C05419=1052.295,341.626,-112.495,173.245,38.864,157.407
C05420=1052.302,341.873,-112.531,173.249,38.868,157.408
C05421=1052.309,342.120,-112.568,173.254,38.872,157.409
C05422=1052.316,342.368,-112.604,173.258,38.877,157.410
C05423=1052.322,342.616,-112.640,173.262,38.881,157.411
C05424=1052.330,342.863,-112.676,173.267,38.886,157.413
C05425=1052.337,343.109,-112.713,173.271,38.890,157.414
C05426=1052.344,343.357,-112.749,173.276,38.894,157.415
C05427=1052.351,343.604,-112.786,173.280,38.899,157.416
C05428=1052.358,343.851,-112.822,173.284,38.904,157.417
C05429=1052.365,344.098,-112.858,173.289,38.908,157.418
C05430=1052.372,344.346,-112.894,173.293,38.913,157.419
C05431=1052.379,344.593,-112.931,173.298,38.917,157.421
C05432=1052.386,344.841,-112.968,173.302,38.921,157.422
C05433=1052.393,345.088,-113.004,173.306,38.926,157.423
C05434=1052.400,345.335,-113.041,173.312,38.931,157.424
C05435=1052.407,345.582,-113.078,173.316,38.935,157.425
C05436=1052.414,345.829,-113.114,173.321,38.939,157.426
C05437=1052.421,346.077,-113.151,173.325,38.944,157.428
C05438=1052.429,346.355,-113.192,173.330,38.949,157.429
C05439=1052.437,346.633,-113.233,173.335,38.954,157.430
C05440=1052.444,346.912,-113.275,173.340,38.959,157.432
C05441=1052.454,347.190,-113.316,173.346,38.964,157.433
C05442=1052.460,347.437,-113.353,173.350,38.969,157.434
C05443=1052.467,347.685,-113.390,173.355,38.973,157.435
C05444=1052.474,347.932,-113.427,173.359,38.978,157.437
C05445=1052.481,348.179,-113.463,173.364,38.982,157.438
C05446=1052.489,348.426,-113.501,173.368,38.987,157.439
C05447=1052.495,348.674,-113.537,173.373,38.992,157.440
C05448=1052.503,348.920,-113.574,173.377,38.996,157.441
C05449=1052.510,349.168,-113.611,173.382,39.001,157.443
C05450=1052.517,349.415,-113.648,173.386,39.005,157.444
C05451=1052.524,349.663,-113.685,173.391,39.010,157.445
C05452=1052.532,349.910,-113.722,173.396,39.015,157.446
C05453=1052.539,350.156,-113.759,173.401,39.019,157.447
C05454=1052.545,350.404,-113.796,173.405,39.024,157.449
C05455=1052.553,350.651,-113.834,173.410,39.028,157.450
C05456=1052.561,350.898,-113.870,173.414,39.033,157.451
C05457=1052.568,351.145,-113.907,173.419,39.038,157.452
C05458=1052.574,351.392,-113.944,173.423,39.043,157.453
C05459=1052.582,351.639,-113.982,173.429,39.047,157.455
C05460=1052.589,351.886,-114.019,173.433,39.052,157.456
C05461=1052.596,352.134,-114.056,173.438,39.057,157.457
C05462=1052.603,352.381,-114.094,173.443,39.062,157.458
C05463=1052.610,352.628,-114.131,173.447,39.066,157.460
C05464=1052.617,352.875,-114.168,173.452,39.071,157.461
C05465=1052.624,353.122,-114.206,173.456,39.076,157.462
C05466=1052.631,353.369,-114.244,173.462,39.081,157.463
C05467=1052.639,353.616,-114.281,173.466,39.086,157.465
C05468=1052.646,353.863,-114.319,173.471,39.090,157.466
C05469=1052.653,354.110,-114.356,173.476,39.095,157.467
C05470=1052.660,354.357,-114.394,173.480,39.100,157.468
C05471=1052.668,354.605,-114.431,173.485,39.105,157.470
C05472=1052.675,354.852,-114.469,173.490,39.109,157.471
C05473=1052.682,355.099,-114.506,173.495,39.114,157.472
C05474=1052.689,355.346,-114.544,173.500,39.119,157.474
C05475=1052.697,355.593,-114.581,173.504,39.124,157.475
C05476=1052.703,355.840,-114.618,173.509,39.129,157.476
C05477=1052.711,356.087,-114.656,173.515,39.134,157.477
C05478=1052.719,356.334,-114.695,173.519,39.139,157.479
C05479=1052.726,356.581,-114.732,173.524,39.144,157.480
C05480=1052.733,356.828,-114.770,173.529,39.148,157.481
C05481=1052.740,357.075,-114.807,173.534,39.153,157.483
C05482=1052.748,357.322,-114.845,173.539,39.158,157.484
C05483=1052.755,357.569,-114.883,173.544,39.163,157.485
C05484=1052.762,357.816,-114.920,173.548,39.168,157.486
C05485=1052.769,358.063,-114.959,173.553,39.173,157.488
C05486=1052.776,358.310,-114.997,173.559,39.178,157.489
C05487=1052.784,358.557,-115.034,173.563,39.183,157.490
C05488=1052.791,358.804,-115.073,173.568,39.188,157.492
C05489=1052.798,359.051,-115.110,173.573,39.193,157.493
C05490=1052.805,359.298,-115.149,173.579,39.198,157.494
C05491=1052.812,359.545,-115.186,173.583,39.203,157.496
C05492=1052.821,359.792,-115.225,173.588,39.208,157.497
C05493=1052.828,360.039,-115.263,173.593,39.213,157.498
C05494=1052.836,360.323,-115.307,173.599,39.219,157.500
C05495=1052.845,360.606,-115.350,173.604,39.224,157.501
C05496=1052.853,360.890,-115.394,173.611,39.230,157.503
C05497=1052.861,361.174,-115.438,173.616,39.236,157.505
C05498=1052.869,361.420,-115.477,173.621,39.241,157.506
C05499=1052.876,361.667,-115.515,173.627,39.246,157.507
C05500=1052.883,361.914,-115.553,173.631,39.251,157.509
C05501=1052.891,362.161,-115.591,173.636,39.257,157.510
C05502=1052.899,362.408,-115.630,173.642,39.262,157.511
C05503=1052.905,362.655,-115.669,173.647,39.267,157.513
C05504=1052.913,362.901,-115.707,173.651,39.272,157.514
C05505=1052.920,363.148,-115.744,173.657,39.277,157.516
C05506=1052.928,363.396,-115.784,173.662,39.282,157.517
C05507=1052.935,363.642,-115.822,173.667,39.287,157.518
C05508=1052.942,363.889,-115.861,173.673,39.293,157.520
C05509=1052.950,364.136,-115.899,173.677,39.298,157.521
C05510=1052.957,364.383,-115.938,173.682,39.303,157.523
C05511=1052.965,364.630,-115.976,173.688,39.309,157.524
C05512=1052.971,364.877,-116.015,173.693,39.314,157.525
C05513=1052.980,365.124,-116.054,173.698,39.319,157.527
C05514=1052.986,365.371,-116.093,173.704,39.324,157.528
C05515=1052.994,365.617,-116.132,173.708,39.330,157.530
C05516=1053.002,365.864,-116.171,173.713,39.335,157.531
C05517=1053.008,366.111,-116.210,173.719,39.340,157.533
C05518=1053.016,366.357,-116.248,173.724,39.346,157.534
C05519=1053.023,366.605,-116.287,173.730,39.351,157.535
C05520=1053.031,366.851,-116.326,173.735,39.356,157.537
C05521=1053.039,367.098,-116.365,173.740,39.362,157.538
C05522=1053.045,367.345,-116.404,173.746,39.367,157.540
C05523=1053.053,367.592,-116.442,173.751,39.373,157.541
C05524=1053.061,367.839,-116.482,173.755,39.378,157.543
C05525=1053.068,368.085,-116.520,173.761,39.383,157.544
C05526=1053.076,368.332,-116.560,173.766,39.389,157.546
C05527=1053.084,368.579,-116.599,173.772,39.394,157.547
C05528=1053.091,368.826,-116.638,173.777,39.399,157.549
C05529=1053.098,369.072,-116.677,173.782,39.405,157.550
C05530=1053.106,369.319,-116.716,173.788,39.410,157.551
C05531=1053.113,369.566,-116.756,173.793,39.415,157.553
C05532=1053.121,369.813,-116.795,173.799,39.421,157.555
C05533=1053.129,370.060,-116.834,173.804,39.427,157.556
C05534=1053.136,370.307,-116.873,173.810,39.432,157.557
C05535=1053.144,370.553,-116.912,173.815,39.437,157.559
C05536=1053.152,370.799,-116.952,173.821,39.443,157.561
C05537=1053.159,371.047,-116.991,173.826,39.449,157.562
C05538=1053.167,371.294,-117.030,173.831,39.454,157.563
C05539=1053.175,371.540,-117.070,173.837,39.460,157.565
C05540=1053.182,371.787,-117.109,173.842,39.465,157.567
C05541=1053.189,372.033,-117.149,173.848,39.471,157.568
C05542=1053.197,372.280,-117.189,173.853,39.477,157.570
C05543=1053.205,372.527,-117.228,173.859,39.482,157.571
C05544=1053.212,372.773,-117.267,173.864,39.488,157.573
C05545=1053.220,373.020,-117.307,173.870,39.494,157.574
C05546=1053.228,373.268,-117.347,173.875,39.500,157.576
C05547=1053.235,373.514,-117.386,173.881,39.505,157.577
C05548=1053.242,373.761,-117.426,173.886,39.511,157.579
C05549=1053.250,374.008,-117.466,173.892,39.517,157.581
C05550=1053.259,374.310,-117.515,173.899,39.524,157.582
C05551=1053.269,374.611,-117.564,173.906,39.531,157.584
C05552=1053.278,374.914,-117.613,173.913,39.538,157.586
C05553=1053.287,375.216,-117.662,173.919,39.544,157.588
C05554=1053.294,375.463,-117.702,173.925,39.550,157.590
C05555=1053.302,375.710,-117.742,173.932,39.556,157.591
C05556=1053.310,375.957,-117.781,173.937,39.562,157.593
C05557=1053.318,376.204,-117.821,173.943,39.568,157.595
C05558=1053.325,376.449,-117.862,173.948,39.574,157.596
C05559=1053.333,376.696,-117.902,173.954,39.580,157.598
C05560=1053.341,376.943,-117.941,173.960,39.586,157.599
C05561=1053.349,377.189,-117.982,173.965,39.591,157.601
C05562=1053.357,377.436,-118.021,173.972,39.597,157.603
C05563=1053.365,377.683,-118.061,173.977,39.603,157.604
C05564=1053.373,377.929,-118.102,173.983,39.609,157.606
C05565=1053.380,378.176,-118.142,173.989,39.615,157.608
C05566=1053.388,378.422,-118.182,173.994,39.621,157.609
C05567=1053.396,378.669,-118.222,174.000,39.627,157.611
C05568=1053.404,378.915,-118.263,174.006,39.633,157.613
C05569=1053.411,379.162,-118.303,174.012,39.639,157.614
C05570=1053.419,379.409,-118.344,174.018,39.645,157.616
C05571=1053.426,379.655,-118.384,174.023,39.650,157.617
C05572=1053.434,379.902,-118.424,174.030,39.656,157.619
C05573=1053.442,380.149,-118.464,174.036,39.663,157.621
C05574=1053.450,380.395,-118.505,174.041,39.668,157.622
C05575=1053.458,380.641,-118.546,174.047,39.675,157.624
C05576=1053.465,380.888,-118.587,174.054,39.681,157.626
C05577=1053.473,381.134,-118.628,174.059,39.687,157.628
C05578=1053.481,381.381,-118.667,174.065,39.693,157.629
C05579=1053.488,381.628,-118.709,174.071,39.699,157.631
C05580=1053.497,381.874,-118.749,174.078,39.706,157.633
C05581=1053.505,382.120,-118.790,174.083,39.711,157.634
C05582=1053.512,382.367,-118.831,174.089,39.718,157.636
C05583=1053.520,382.613,-118.872,174.095,39.724,157.638
C05584=1053.528,382.860,-118.913,174.101,39.731,157.640
C05585=1053.536,383.107,-118.954,174.107,39.736,157.641
C05586=1053.544,383.353,-118.995,174.113,39.743,157.643
C05587=1053.552,383.599,-119.035,174.120,39.749,157.645
C05588=1053.559,383.846,-119.077,174.125,39.755,157.647
C05589=1053.567,384.092,-119.117,174.131,39.762,157.649
C05590=1053.575,384.338,-119.159,174.138,39.768,157.650
C05591=1053.583,384.585,-119.200,174.144,39.774,157.652
C05592=1053.591,384.831,-119.241,174.150,39.780,157.654
C05593=1053.599,385.078,-119.282,174.156,39.787,157.655
C05594=1053.607,385.324,-119.323,174.162,39.793,157.657
C05595=1053.615,385.570,-119.364,174.169,39.799,157.659
C05596=1053.623,385.817,-119.406,174.175,39.806,157.661
C05597=1053.631,386.063,-119.446,174.181,39.813,157.663
C05598=1053.639,386.309,-119.488,174.187,39.819,157.665
C05599=1053.647,386.556,-119.529,174.193,39.825,157.666
C05600=1053.655,386.802,-119.570,174.200,39.832,157.668
C05601=1053.663,387.049,-119.612,174.206,39.838,157.670
C05602=1053.672,387.295,-119.653,174.213,39.845,157.672
C05603=1053.679,387.542,-119.695,174.218,39.851,157.674
C05604=1053.687,387.787,-119.736,174.225,39.857,157.675
C05605=1053.695,388.035,-119.778,174.231,39.864,157.677
C05606=1053.704,388.284,-119.819,174.238,39.871,157.679
C05607=1053.712,388.534,-119.861,174.244,39.877,157.681
C05608=1053.721,388.784,-119.904,174.251,39.884,157.683
C05609=1053.728,389.034,-119.946,174.258,39.891,157.685
C05610=1053.737,389.281,-119.987,174.264,39.897,157.687
C05611=1053.745,389.527,-120.029,174.271,39.904,157.689
C05612=1053.753,389.773,-120.071,174.277,39.911,157.691
C05613=1053.761,390.019,-120.113,174.283,39.917,157.692
C05614=1053.769,390.266,-120.154,174.289,39.924,157.694
C05615=1053.777,390.512,-120.196,174.296,39.931,157.696
C05616=1053.785,390.758,-120.238,174.302,39.937,157.698
C05617=1053.793,391.005,-120.280,174.309,39.944,157.700
C05618=1053.801,391.250,-120.322,174.315,39.951,157.702
C05619=1053.810,391.497,-120.364,174.322,39.957,157.704
C05620=1053.818,391.744,-120.406,174.329,39.964,157.706
C05621=1053.826,391.990,-120.448,174.335,39.971,157.708
C05622=1053.835,392.235,-120.490,174.342,39.978,157.710
C05623=1053.843,392.481,-120.532,174.348,39.985,157.712
C05624=1053.851,392.728,-120.575,174.355,39.991,157.714
C05625=1053.859,392.975,-120.617,174.362,39.998,157.716
C05626=1053.870,393.304,-120.674,174.371,40.008,157.718
C05627=1053.881,393.636,-120.730,174.380,40.017,157.721
C05628=1053.892,393.966,-120.787,174.389,40.027,157.724
C05629=1053.903,394.297,-120.844,174.398,40.035,157.726
C05630=1053.911,394.543,-120.887,174.405,40.043,157.728
C05631=1053.919,394.789,-120.929,174.411,40.050,157.730
C05632=1053.928,395.035,-120.972,174.418,40.057,157.732
C05633=1053.936,395.282,-121.014,174.425,40.064,157.734
C05634=1053.945,395.527,-121.056,174.432,40.071,157.736
C05635=1053.953,395.774,-121.099,174.439,40.078,157.738
C05636=1053.961,396.020,-121.142,174.446,40.085,157.741
C05637=1053.970,396.266,-121.185,174.453,40.092,157.742
C05638=1053.978,396.512,-121.227,174.459,40.099,157.745
C05639=1053.986,396.758,-121.270,174.466,40.107,157.747
C05640=1053.994,397.004,-121.313,174.473,40.113,157.749
C05641=1054.003,397.251,-121.355,174.480,40.121,157.751
C05642=1054.011,397.497,-121.398,174.488,40.128,157.753
C05643=1054.020,397.743,-121.441,174.494,40.135,157.755
C05644=1054.028,397.989,-121.484,174.501,40.143,157.757
C05645=1054.037,398.235,-121.527,174.508,40.150,157.759
C05646=1054.044,398.481,-121.571,174.515,40.157,157.761
C05647=1054.053,398.727,-121.614,174.523,40.164,157.764
C05648=1054.061,398.973,-121.657,174.529,40.172,157.766
C05649=1054.070,399.219,-121.700,174.536,40.179,157.768
C05650=1054.078,399.465,-121.743,174.543,40.186,157.770
C05651=1054.087,399.711,-121.786,174.550,40.194,157.772
C05652=1054.095,399.957,-121.829,174.558,40.201,157.774
C05653=1054.104,400.203,-121.872,174.565,40.209,157.776
C05654=1054.112,400.450,-121.915,174.572,40.216,157.779
C05655=1054.120,400.696,-121.959,174.579,40.223,157.781
C05656=1054.129,400.941,-122.002,174.587,40.231,157.783
C05657=1054.137,401.187,-122.045,174.594,40.238,157.785
C05658=1054.146,401.433,-122.088,174.601,40.246,157.787
C05659=1054.155,401.680,-122.132,174.608,40.253,157.789
C05660=1054.163,401.926,-122.176,174.615,40.261,157.792
C05661=1054.172,402.172,-122.219,174.622,40.268,157.794
C05662=1054.184,402.524,-122.281,174.634,40.279,157.797
C05663=1054.196,402.877,-122.344,174.644,40.290,157.800
C05664=1054.209,403.230,-122.407,174.655,40.302,157.804
C05665=1054.221,403.582,-122.470,174.665,40.313,157.807
C05666=1054.229,403.828,-122.513,174.672,40.320,157.809
C05667=1054.239,404.074,-122.557,174.680,40.328,157.811
C05668=1054.247,404.320,-122.601,174.687,40.336,157.814
C05669=1054.255,404.566,-122.644,174.695,40.344,157.816
C05670=1054.264,404.812,-122.689,174.702,40.351,157.818
C05671=1054.273,405.058,-122.733,174.710,40.359,157.821
C05672=1054.281,405.303,-122.777,174.718,40.367,157.823
C05673=1054.290,405.550,-122.821,174.726,40.375,157.825
C05674=1054.298,405.795,-122.866,174.733,40.383,157.828
C05675=1054.308,406.041,-122.910,174.741,40.391,157.830
C05676=1054.316,406.287,-122.954,174.748,40.399,157.832
C05677=1054.324,406.533,-122.998,174.756,40.407,157.835
C05678=1054.333,406.779,-123.043,174.763,40.415,157.837
C05679=1054.341,407.025,-123.087,174.772,40.423,157.839
C05680=1054.351,407.271,-123.131,174.779,40.431,157.842
C05681=1054.359,407.517,-123.175,174.787,40.439,157.844
C05682=1054.368,407.763,-123.220,174.794,40.447,157.847
C05683=1054.377,408.008,-123.265,174.802,40.455,157.849
C05684=1054.385,408.254,-123.309,174.811,40.463,157.852
C05685=1054.395,408.501,-123.353,174.818,40.471,157.854
C05686=1054.403,408.746,-123.398,174.826,40.479,157.856
C05687=1054.412,408.992,-123.443,174.833,40.488,157.859
C05688=1054.421,409.238,-123.487,174.842,40.496,157.861
C05689=1054.430,409.483,-123.532,174.850,40.504,157.864
C05690=1054.438,409.730,-123.577,174.857,40.512,157.866
C05691=1054.448,409.975,-123.622,174.866,40.520,157.869
C05692=1054.456,410.221,-123.666,174.874,40.529,157.871
C05693=1054.466,410.467,-123.711,174.881,40.537,157.874
C05694=1054.474,410.713,-123.756,174.890,40.546,157.876
C05695=1054.483,410.959,-123.801,174.898,40.554,157.879
C05696=1054.493,411.204,-123.846,174.906,40.562,157.881
C05697=1054.501,411.450,-123.891,174.914,40.571,157.884
C05698=1054.510,411.696,-123.936,174.922,40.579,157.886
C05699=1054.520,411.941,-123.980,174.931,40.587,157.889
C05700=1054.529,412.187,-124.026,174.938,40.596,157.891
C05701=1054.538,412.433,-124.071,174.947,40.604,157.894
C05702=1054.547,412.679,-124.117,174.955,40.613,157.896
C05703=1054.556,412.924,-124.162,174.964,40.621,157.899
C05704=1054.565,413.170,-124.207,174.972,40.630,157.902
C05705=1054.574,413.416,-124.252,174.980,40.638,157.904
C05706=1054.583,413.662,-124.298,174.988,40.647,157.907
C05707=1054.592,413.908,-124.343,174.997,40.656,157.909
C05708=1054.601,414.154,-124.389,175.005,40.664,157.912
C05709=1054.610,414.399,-124.434,175.014,40.673,157.915
C05710=1054.619,414.645,-124.479,175.022,40.682,157.917
C05711=1054.629,414.890,-124.526,175.031,40.691,157.920
C05712=1054.638,415.136,-124.571,175.040,40.699,157.923
C05713=1054.647,415.382,-124.616,175.048,40.708,157.925
C05714=1054.656,415.627,-124.663,175.057,40.717,157.928
C05715=1054.665,415.873,-124.708,175.066,40.726,157.931
C05716=1054.674,416.118,-124.754,175.074,40.735,157.934
C05717=1054.683,416.364,-124.800,175.083,40.744,157.936
C05718=1054.697,416.723,-124.867,175.095,40.756,157.940
C05719=1054.711,417.081,-124.934,175.108,40.770,157.944
C05720=1054.724,417.440,-125.001,175.121,40.783,157.948
C05721=1054.738,417.798,-125.068,175.133,40.796,157.952
C05722=1054.747,418.043,-125.114,175.142,40.805,157.955
C05723=1054.756,418.289,-125.160,175.152,40.814,157.958
C05724=1054.766,418.535,-125.207,175.161,40.823,157.961
C05725=1054.776,418.780,-125.253,175.170,40.833,157.964
C05726=1054.785,419.026,-125.298,175.178,40.842,157.967
C05727=1054.794,419.272,-125.345,175.187,40.851,157.969
C05728=1054.803,419.517,-125.392,175.196,40.860,157.972
C05729=1054.813,419.763,-125.438,175.205,40.869,157.975
C05730=1054.822,420.008,-125.485,175.215,40.879,157.978
C05731=1054.832,420.253,-125.531,175.224,40.888,157.981
C05732=1054.841,420.499,-125.578,175.233,40.897,157.984
C05733=1054.851,420.745,-125.625,175.242,40.906,157.987
C05734=1054.860,420.989,-125.672,175.252,40.916,157.990
C05735=1054.869,421.235,-125.718,175.261,40.925,157.992
C05736=1054.879,421.481,-125.765,175.269,40.935,157.995
C05737=1054.888,421.725,-125.812,175.278,40.944,157.998
C05738=1054.898,421.972,-125.859,175.288,40.954,158.001
C05739=1054.908,422.217,-125.906,175.298,40.963,158.004
C05740=1054.917,422.462,-125.952,175.307,40.973,158.007
C05741=1054.926,422.708,-126.000,175.317,40.983,158.010
C05742=1054.936,422.952,-126.047,175.326,40.992,158.013
C05743=1054.946,423.198,-126.093,175.335,41.002,158.016
C05744=1054.955,423.444,-126.141,175.345,41.011,158.019
C05745=1054.965,423.688,-126.188,175.354,41.021,158.022
C05746=1054.974,423.935,-126.235,175.364,41.031,158.026
C05747=1054.984,424.180,-126.282,175.373,41.041,158.029
C05748=1054.995,424.425,-126.329,175.384,41.051,158.032
C05749=1055.004,424.671,-126.377,175.393,41.060,158.035
C05750=1055.014,424.915,-126.424,175.403,41.070,158.038
C05751=1055.023,425.161,-126.472,175.412,41.080,158.041
C05752=1055.033,425.406,-126.519,175.422,41.090,158.044
C05753=1055.043,425.651,-126.566,175.432,41.100,158.047
C05754=1055.053,425.897,-126.614,175.442,41.110,158.051
C05755=1055.063,426.142,-126.662,175.451,41.120,158.054
C05756=1055.073,426.387,-126.710,175.462,41.130,158.057
C05757=1055.082,426.633,-126.758,175.472,41.140,158.060
C05758=1055.092,426.877,-126.805,175.481,41.150,158.063
C05759=1055.102,427.122,-126.853,175.492,41.160,158.066
C05760=1055.112,427.368,-126.900,175.502,41.170,158.070
C05761=1055.122,427.613,-126.949,175.511,41.180,158.073
C05762=1055.131,427.858,-126.997,175.522,41.190,158.076
C05763=1055.142,428.103,-127.045,175.532,41.201,158.080
C05764=1055.151,428.348,-127.093,175.542,41.211,158.083
C05765=1055.161,428.594,-127.141,175.552,41.221,158.086
C05766=1055.172,428.839,-127.189,175.563,41.232,158.089
C05767=1055.182,429.084,-127.238,175.573,41.242,158.093
C05768=1055.191,429.329,-127.286,175.584,41.252,158.096
C05769=1055.202,429.574,-127.333,175.593,41.262,158.099
C05770=1055.211,429.819,-127.382,175.604,41.273,158.103
C05771=1055.222,430.065,-127.431,175.615,41.283,158.106
C05772=1055.231,430.310,-127.479,175.625,41.294,158.110
C05773=1055.242,430.554,-127.527,175.636,41.305,158.113
C05774=1055.257,430.935,-127.603,175.652,41.321,158.118
C05775=1055.273,431.316,-127.679,175.668,41.337,158.124
C05776=1055.289,431.696,-127.755,175.686,41.354,158.129
C05777=1055.304,432.077,-127.831,175.702,41.371,158.135
C05778=1055.314,432.321,-127.880,175.713,41.381,158.138
C05779=1055.325,432.567,-127.929,175.724,41.392,158.141
C05780=1055.335,432.811,-127.978,175.735,41.403,158.145
C05781=1055.345,433.057,-128.027,175.745,41.414,158.149
C05782=1055.355,433.301,-128.076,175.756,41.425,158.152
C05783=1055.366,433.547,-128.125,175.767,41.436,158.156
C05784=1055.376,433.791,-128.174,175.779,41.447,158.159
C05785=1055.387,434.036,-128.223,175.790,41.458,158.163
C05786=1055.397,434.280,-128.273,175.801,41.469,158.166
C05787=1055.407,434.526,-128.321,175.812,41.480,158.170
C05788=1055.418,434.771,-128.371,175.823,41.491,158.174
C05789=1055.428,435.015,-128.420,175.835,41.502,158.177
C05790=1055.439,435.260,-128.470,175.846,41.514,158.181
C05791=1055.449,435.505,-128.519,175.857,41.524,158.185
C05792=1055.460,435.750,-128.569,175.869,41.536,158.189
C05793=1055.470,435.995,-128.618,175.880,41.547,158.192
C05794=1055.481,436.239,-128.669,175.891,41.558,158.196
C05795=1055.492,436.484,-128.718,175.903,41.570,158.200
C05796=1055.503,436.729,-128.768,175.914,41.581,158.203
C05797=1055.513,436.974,-128.817,175.926,41.593,158.207
C05798=1055.524,437.218,-128.867,175.938,41.604,158.211
C05799=1055.534,437.463,-128.917,175.949,41.615,158.215
C05800=1055.544,437.708,-128.968,175.961,41.627,158.219
C05801=1055.555,437.953,-129.018,175.973,41.639,158.223
C05802=1055.566,438.197,-129.068,175.985,41.650,158.226
C05803=1055.577,438.442,-129.118,175.997,41.662,158.230
C05804=1055.588,438.686,-129.169,176.008,41.673,158.234
C05805=1055.598,438.932,-129.219,176.021,41.685,158.238
C05806=1055.609,439.176,-129.269,176.033,41.697,158.242
C05807=1055.620,439.420,-129.319,176.044,41.708,158.246
C05808=1055.631,439.665,-129.370,176.057,41.721,158.250
C05809=1055.641,439.910,-129.421,176.069,41.732,158.254
C05810=1055.652,440.154,-129.471,176.081,41.744,158.258
C05811=1055.663,440.398,-129.521,176.093,41.756,158.262
C05812=1055.673,440.643,-129.572,176.106,41.768,158.266
C05813=1055.685,440.888,-129.624,176.118,41.780,158.270
C05814=1055.696,441.132,-129.674,176.131,41.792,158.274
C05815=1055.706,441.377,-129.725,176.143,41.804,158.278
C05816=1055.718,441.621,-129.776,176.155,41.816,158.283
C05817=1055.729,441.866,-129.827,176.167,41.828,158.287
C05818=1055.740,442.110,-129.878,176.180,41.840,158.291
C05819=1055.751,442.354,-129.929,176.193,41.853,158.295
C05820=1055.762,442.599,-129.981,176.205,41.865,158.299
C05821=1055.773,442.844,-130.031,176.218,41.877,158.303
C05822=1055.784,443.088,-130.083,176.231,41.890,158.308
C05823=1055.795,443.332,-130.134,176.244,41.902,158.312
C05824=1055.806,443.576,-130.186,176.257,41.914,158.316
C05825=1055.818,443.821,-130.237,176.270,41.927,158.320
C05826=1055.828,444.065,-130.289,176.283,41.939,158.325
C05827=1055.840,444.310,-130.340,176.296,41.952,158.329
C05828=1055.851,444.554,-130.392,176.309,41.964,158.333
C05829=1055.863,444.798,-130.443,176.322,41.977,158.338
C05830=1055.880,445.158,-130.519,176.342,41.996,158.344
C05831=1055.896,445.517,-130.595,176.361,42.015,158.351
C05832=1055.913,445.876,-130.671,176.381,42.033,158.357
C05833=1055.929,446.235,-130.748,176.401,42.052,158.364
C05834=1055.941,446.479,-130.800,176.414,42.065,158.368
C05835=1055.953,446.722,-130.852,176.428,42.078,158.373
C05836=1055.966,446.965,-130.903,176.442,42.090,158.377
C05837=1055.978,447.210,-130.954,176.455,42.103,158.381
C05838=1055.992,447.453,-131.004,176.470,42.115,158.386
C05839=1056.006,447.697,-131.053,176.483,42.127,158.390
C05840=1056.022,447.941,-131.103,176.497,42.139,158.394
C05841=1056.038,448.186,-131.151,176.511,42.151,158.399
C05842=1056.055,448.430,-131.199,176.525,42.162,158.403
C05843=1056.073,448.675,-131.246,176.539,42.174,158.407
C05844=1056.091,448.919,-131.294,176.553,42.185,158.411
C05845=1056.111,449.164,-131.339,176.568,42.196,158.415
C05846=1056.131,449.410,-131.385,176.583,42.207,158.419
C05847=1056.153,449.654,-131.430,176.597,42.217,158.423
C05848=1056.174,449.899,-131.475,176.612,42.228,158.427
C05849=1056.197,450.146,-131.519,176.626,42.238,158.431
C05850=1055.873,450.163,-131.806,176.624,42.342,158.460
C05851=1055.851,449.918,-131.763,176.609,42.332,158.456
C05852=1055.829,449.673,-131.718,176.594,42.321,158.452
C05853=1055.808,449.427,-131.674,176.579,42.311,158.448
C05854=1055.787,449.182,-131.627,176.565,42.300,158.444
C05855=1055.768,448.937,-131.581,176.550,42.289,158.440
C05856=1055.749,448.693,-131.534,176.537,42.278,158.436
C05857=1055.731,448.447,-131.488,176.523,42.267,158.432
C05858=1055.714,448.204,-131.439,176.507,42.256,158.428
C05859=1055.697,447.959,-131.391,176.493,42.244,158.424
C05860=1055.681,447.715,-131.342,176.480,42.232,158.419
C05861=1055.666,447.471,-131.292,176.466,42.220,158.415
C05862=1055.652,447.227,-131.242,176.451,42.208,158.411
C05863=1055.640,446.983,-131.192,176.438,42.195,158.406
C05864=1055.627,446.739,-131.140,176.424,42.183,158.402
C05865=1055.615,446.496,-131.088,176.410,42.170,158.397
C05866=1055.604,446.253,-131.037,176.397,42.157,158.393
C05867=1055.587,445.913,-130.965,176.378,42.140,158.387
C05868=1055.571,445.572,-130.892,176.360,42.122,158.380
C05869=1055.555,445.232,-130.819,176.340,42.104,158.374
C05870=1055.539,444.893,-130.747,176.322,42.087,158.368
C05871=1055.528,444.648,-130.695,176.308,42.074,158.364
C05872=1055.517,444.404,-130.644,176.295,42.062,158.359
C05873=1055.506,444.159,-130.592,176.282,42.049,158.355
C05874=1055.494,443.915,-130.541,176.269,42.037,158.351
C05875=1055.483,443.670,-130.489,176.256,42.024,158.346
C05876=1055.472,443.427,-130.438,176.243,42.012,158.342
C05877=1055.461,443.182,-130.386,176.230,41.999,158.338
C05878=1055.449,442.938,-130.335,176.217,41.987,158.334
C05879=1055.439,442.693,-130.284,176.204,41.975,158.329
C05880=1055.427,442.449,-130.233,176.192,41.963,158.325
C05881=1055.416,442.204,-130.181,176.179,41.950,158.321
C05882=1055.405,441.959,-130.131,176.166,41.938,158.317
C05883=1055.394,441.716,-130.080,176.154,41.926,158.313
C05884=1055.383,441.470,-130.028,176.141,41.914,158.309
C05885=1055.372,441.226,-129.977,176.128,41.902,158.304
C05886=1055.361,440.982,-129.927,176.116,41.890,158.301
C05887=1055.351,440.737,-129.876,176.103,41.878,158.296
C05888=1055.339,440.492,-129.825,176.091,41.866,158.292
C05889=1055.328,440.248,-129.774,176.079,41.854,158.288
C05890=1055.318,440.004,-129.723,176.067,41.843,158.284
C05891=1055.307,439.759,-129.673,176.054,41.831,158.280
C05892=1055.296,439.515,-129.623,176.042,41.819,158.276
C05893=1055.285,439.270,-129.572,176.030,41.807,158.272
C05894=1055.274,439.026,-129.521,176.018,41.796,158.268
C05895=1055.263,438.781,-129.471,176.005,41.784,158.264
C05896=1055.252,438.536,-129.420,175.993,41.772,158.260
C05897=1055.241,438.291,-129.371,175.982,41.761,158.257
C05898=1055.231,438.047,-129.320,175.969,41.749,158.253
C05899=1055.221,437.802,-129.270,175.958,41.738,158.249
C05900=1055.210,437.557,-129.220,175.946,41.726,158.245
C05901=1055.199,437.313,-129.170,175.934,41.715,158.241
C05902=1055.188,437.068,-129.120,175.922,41.704,158.237
C05903=1055.177,436.824,-129.070,175.910,41.692,158.233
C05904=1055.167,436.578,-129.020,175.899,41.680,158.230
C05905=1055.156,436.333,-128.971,175.888,41.669,158.226
C05906=1055.145,436.088,-128.921,175.876,41.658,158.222
C05907=1055.134,435.844,-128.871,175.865,41.647,158.218
C05908=1055.124,435.600,-128.822,175.853,41.635,158.215
C05909=1055.114,435.355,-128.772,175.841,41.625,158.211
C05910=1055.103,435.109,-128.722,175.830,41.613,158.207
C05911=1055.092,434.864,-128.673,175.818,41.603,158.204
C05912=1055.082,434.620,-128.624,175.807,41.591,158.200
C05913=1055.071,434.375,-128.574,175.796,41.581,158.196
C05914=1055.061,434.131,-128.525,175.784,41.569,158.193
C05915=1055.051,433.885,-128.476,175.773,41.558,158.189
C05916=1055.040,433.640,-128.426,175.763,41.547,158.185
C05917=1055.030,433.396,-128.377,175.752,41.537,158.182
C05918=1055.020,433.151,-128.327,175.741,41.526,158.178
C05919=1055.010,432.906,-128.279,175.730,41.515,158.175
C05920=1054.999,432.660,-128.229,175.718,41.504,158.171
C05921=1054.989,432.416,-128.181,175.707,41.493,158.168
C05922=1054.978,432.171,-128.132,175.696,41.482,158.164
C05923=1054.963,431.788,-128.056,175.680,41.466,158.159
C05924=1054.947,431.406,-127.979,175.663,41.449,158.153
C05925=1054.931,431.023,-127.903,175.646,41.432,158.148
C05926=1054.916,430.641,-127.827,175.630,41.416,158.142
C05927=1054.906,430.397,-127.778,175.619,41.406,158.139
C05928=1054.895,430.151,-127.729,175.608,41.395,158.135
C05929=1054.885,429.906,-127.681,175.598,41.384,158.132
C05930=1054.875,429.661,-127.633,175.587,41.374,158.129
C05931=1054.865,429.416,-127.585,175.576,41.364,158.126
C05932=1054.855,429.170,-127.536,175.567,41.354,158.122
C05933=1054.845,428.925,-127.488,175.556,41.343,158.119
C05934=1054.835,428.680,-127.440,175.546,41.333,158.115
C05935=1054.825,428.435,-127.391,175.535,41.323,158.112
C05936=1054.815,428.190,-127.344,175.525,41.312,158.109
C05937=1054.805,427.945,-127.295,175.515,41.302,158.106
C05938=1054.795,427.700,-127.247,175.505,41.292,158.102
C05939=1054.785,427.455,-127.200,175.494,41.282,158.099
C05940=1054.775,427.210,-127.151,175.484,41.272,158.096
C05941=1054.765,426.965,-127.104,175.475,41.262,158.093
C05942=1054.755,426.720,-127.055,175.464,41.252,158.089
C05943=1054.746,426.474,-127.007,175.454,41.241,158.086
C05944=1054.736,426.229,-126.960,175.444,41.231,158.083
C05945=1054.726,425.984,-126.912,175.434,41.222,158.080
C05946=1054.716,425.738,-126.865,175.424,41.211,158.076
C05947=1054.706,425.493,-126.817,175.415,41.202,158.073
C05948=1054.696,425.248,-126.769,175.404,41.192,158.070
C05949=1054.686,425.002,-126.722,175.394,41.182,158.067
C05950=1054.677,424.757,-126.674,175.385,41.172,158.064
C05951=1054.667,424.512,-126.628,175.375,41.162,158.061
C05952=1054.658,424.267,-126.580,175.365,41.153,158.058
C05953=1054.647,424.021,-126.533,175.356,41.143,158.055
C05954=1054.637,423.776,-126.485,175.346,41.133,158.052
C05955=1054.628,423.531,-126.438,175.337,41.124,158.049
C05956=1054.618,423.285,-126.391,175.327,41.114,158.046
C05957=1054.608,423.040,-126.344,175.318,41.105,158.043
C05958=1054.599,422.794,-126.296,175.307,41.095,158.040
C05959=1054.589,422.549,-126.250,175.298,41.086,158.037
C05960=1054.579,422.304,-126.203,175.288,41.076,158.034
C05961=1054.570,422.059,-126.156,175.279,41.067,158.031
C05962=1054.561,421.813,-126.109,175.270,41.057,158.027
C05963=1054.551,421.567,-126.061,175.260,41.047,158.024
C05964=1054.542,421.322,-126.015,175.251,41.038,158.022
C05965=1054.532,421.077,-125.968,175.242,41.029,158.019
C05966=1054.523,420.831,-125.921,175.232,41.019,158.016
C05967=1054.513,420.585,-125.875,175.223,41.010,158.013
C05968=1054.504,420.340,-125.829,175.214,41.001,158.010
C05969=1054.494,420.095,-125.781,175.205,40.991,158.007
C05970=1054.485,419.849,-125.735,175.196,40.982,158.004
C05971=1054.476,419.604,-125.688,175.187,40.973,158.001
C05972=1054.466,419.358,-125.642,175.178,40.964,157.998
C05973=1054.457,419.113,-125.596,175.169,40.955,157.995
C05974=1054.447,418.867,-125.549,175.160,40.945,157.993
C05975=1054.438,418.622,-125.503,175.150,40.936,157.990
C05976=1054.428,418.376,-125.457,175.141,40.927,157.987
C05977=1054.418,418.131,-125.411,175.132,40.918,157.984
C05978=1054.410,417.885,-125.364,175.124,40.909,157.981
C05979=1054.395,417.525,-125.297,175.110,40.896,157.977
C05980=1054.382,417.164,-125.230,175.098,40.883,157.973
C05981=1054.368,416.804,-125.161,175.085,40.870,157.969
C05982=1054.354,416.443,-125.094,175.072,40.857,157.965
C05983=1054.345,416.197,-125.049,175.063,40.848,157.962
C05984=1054.336,415.952,-125.002,175.054,40.839,157.960
C05985=1054.327,415.706,-124.957,175.046,40.830,157.957
C05986=1054.318,415.461,-124.911,175.037,40.821,157.954
C05987=1054.309,415.215,-124.865,175.029,40.812,157.951
C05988=1054.300,414.970,-124.819,175.020,40.804,157.949
C05989=1054.291,414.724,-124.774,175.011,40.795,157.946
C05990=1054.282,414.478,-124.728,175.003,40.787,157.944
C05991=1054.272,414.233,-124.682,174.994,40.778,157.941
C05992=1054.263,413.987,-124.637,174.986,40.769,157.938
C05993=1054.254,413.741,-124.591,174.977,40.761,157.936
C05994=1054.245,413.495,-124.546,174.969,40.752,157.933
C05995=1054.236,413.250,-124.501,174.961,40.743,157.930
C05996=1054.227,413.003,-124.455,174.952,40.735,157.928
C05997=1054.217,412.758,-124.410,174.944,40.726,157.925
C05998=1054.208,412.512,-124.365,174.935,40.718,157.922
C05999=1054.199,412.266,-124.319,174.927,40.709,157.920
C06000=1054.191,412.021,-124.274,174.918,40.701,157.917
C06001=1054.181,411.775,-124.229,174.911,40.693,157.915
C06002=1054.172,411.529,-124.184,174.903,40.684,157.912
C06003=1054.163,411.283,-124.139,174.894,40.676,157.910
C06004=1054.154,411.038,-124.094,174.886,40.668,157.907
C06005=1054.145,410.792,-124.049,174.878,40.659,157.905
C06006=1054.136,410.545,-124.004,174.870,40.651,157.902
C06007=1054.127,410.300,-123.960,174.861,40.643,157.900
C06008=1054.118,410.055,-123.914,174.853,40.634,157.897
C06009=1054.109,409.808,-123.870,174.846,40.626,157.895
C06010=1054.100,409.563,-123.825,174.837,40.618,157.892
C06011=1054.091,409.317,-123.780,174.829,40.610,157.890
C06012=1054.082,409.071,-123.736,174.822,40.601,157.887
C06013=1054.073,408.825,-123.691,174.813,40.593,157.885
C06014=1054.065,408.580,-123.646,174.805,40.586,157.882
C06015=1054.055,408.334,-123.602,174.798,40.577,157.880
C06016=1054.047,408.087,-123.557,174.790,40.569,157.877
C06017=1054.038,407.842,-123.513,174.781,40.561,157.875
C06018=1054.029,407.596,-123.468,174.774,40.553,157.873
C06019=1054.021,407.350,-123.424,174.766,40.545,157.870
C06020=1054.011,407.104,-123.379,174.759,40.537,157.868
C06021=1054.003,406.858,-123.335,174.751,40.529,157.865
C06022=1053.994,406.612,-123.291,174.743,40.521,157.863
C06023=1053.986,406.367,-123.246,174.735,40.513,157.861
C06024=1053.977,406.121,-123.201,174.727,40.505,157.858
C06025=1053.968,405.875,-123.158,174.720,40.497,157.856
C06026=1053.959,405.629,-123.113,174.712,40.489,157.854
C06027=1053.951,405.383,-123.069,174.705,40.481,157.851
C06028=1053.943,405.137,-123.025,174.696,40.474,157.849
C06029=1053.933,404.891,-122.981,174.689,40.466,157.847
C06030=1053.925,404.645,-122.937,174.681,40.458,157.844
C06031=1053.916,404.399,-122.893,174.674,40.450,157.842
C06032=1053.908,404.153,-122.849,174.666,40.442,157.840
C06033=1053.899,403.907,-122.806,174.659,40.435,157.837
C06034=1053.890,403.661,-122.761,174.652,40.427,157.835
C06035=1053.878,403.307,-122.698,174.641,40.416,157.832
C06036=1053.866,402.952,-122.635,174.630,40.405,157.829
C06037=1053.853,402.598,-122.572,174.619,40.394,157.825
C06038=1053.841,402.243,-122.509,174.609,40.383,157.822
C06039=1053.832,401.997,-122.466,174.601,40.375,157.820
C06040=1053.824,401.752,-122.422,174.594,40.368,157.818
C06041=1053.815,401.506,-122.379,174.587,40.360,157.815
C06042=1053.807,401.260,-122.335,174.579,40.353,157.813
C06043=1053.798,401.013,-122.292,174.572,40.345,157.811
C06044=1053.789,400.767,-122.249,174.565,40.338,157.809
C06045=1053.781,400.521,-122.205,174.557,40.331,157.807
C06046=1053.772,400.276,-122.161,174.550,40.323,157.804
C06047=1053.764,400.030,-122.118,174.543,40.316,157.802
C06048=1053.755,399.783,-122.075,174.536,40.309,157.800
C06049=1053.747,399.537,-122.032,174.529,40.301,157.798
C06050=1053.738,399.291,-121.989,174.522,40.294,157.796
C06051=1053.730,399.045,-121.946,174.515,40.287,157.794
C06052=1053.721,398.799,-121.903,174.507,40.279,157.792
C06053=1053.713,398.553,-121.860,174.500,40.272,157.789
C06054=1053.705,398.307,-121.817,174.493,40.265,157.787
C06055=1053.697,398.061,-121.774,174.486,40.258,157.785
C06056=1053.688,397.815,-121.731,174.479,40.250,157.783
C06057=1053.680,397.569,-121.688,174.472,40.243,157.781
C06058=1053.671,397.323,-121.645,174.465,40.236,157.779
C06059=1053.663,397.077,-121.602,174.458,40.228,157.777
C06060=1053.654,396.830,-121.559,174.451,40.222,157.775
C06061=1053.646,396.584,-121.516,174.445,40.214,157.773
C06062=1053.638,396.338,-121.474,174.437,40.207,157.771
C06063=1053.630,396.092,-121.431,174.430,40.200,157.769
C06064=1053.621,395.846,-121.388,174.423,40.193,157.766
C06065=1053.613,395.600,-121.345,174.417,40.186,157.764
C06066=1053.604,395.353,-121.303,174.410,40.179,157.762
C06067=1053.596,395.108,-121.261,174.403,40.172,157.760
C06068=1053.588,394.861,-121.218,174.396,40.165,157.758
C06069=1053.579,394.615,-121.175,174.389,40.158,157.756
C06070=1053.571,394.369,-121.133,174.382,40.151,157.754
C06071=1053.563,394.123,-121.090,174.375,40.144,157.752
C06072=1053.555,393.877,-121.048,174.369,40.137,157.750
C06073=1053.546,393.630,-121.006,174.362,40.130,157.748
C06074=1053.538,393.385,-120.964,174.355,40.124,157.746
C06075=1053.530,393.138,-120.922,174.349,40.117,157.744
C06076=1053.522,392.891,-120.879,174.342,40.110,157.742
C06077=1053.514,392.646,-120.837,174.335,40.103,157.740
C06078=1053.506,392.399,-120.794,174.329,40.096,157.738
C06079=1053.497,392.153,-120.753,174.322,40.089,157.736
C06080=1053.489,391.907,-120.711,174.315,40.083,157.735
C06081=1053.481,391.660,-120.668,174.309,40.076,157.733
C06082=1053.473,391.415,-120.627,174.302,40.069,157.731
C06083=1053.464,391.168,-120.585,174.296,40.062,157.729
C06084=1053.457,390.922,-120.543,174.289,40.055,157.727
C06085=1053.448,390.676,-120.501,174.282,40.049,157.725
C06086=1053.440,390.430,-120.459,174.276,40.042,157.723
C06087=1053.432,390.183,-120.417,174.269,40.035,157.721
C06088=1053.424,389.937,-120.375,174.263,40.029,157.719
C06089=1053.416,389.691,-120.333,174.256,40.022,157.717
C06090=1053.408,389.445,-120.291,174.250,40.015,157.715
C06091=1053.396,389.109,-120.235,174.240,40.007,157.713
C06092=1053.385,388.772,-120.178,174.232,39.998,157.710
C06093=1053.374,388.436,-120.121,174.223,39.989,157.708
C06094=1053.363,388.099,-120.064,174.215,39.980,157.705
C06095=1053.355,387.852,-120.023,174.208,39.973,157.703
C06096=1053.346,387.606,-119.981,174.202,39.967,157.701
C06097=1053.339,387.360,-119.940,174.195,39.961,157.700
C06098=1053.330,387.114,-119.898,174.189,39.954,157.698
C06099=1053.323,386.867,-119.857,174.182,39.948,157.696
C06100=1053.314,386.621,-119.815,174.176,39.941,157.694
C06101=1053.306,386.374,-119.775,174.171,39.935,157.692
C06102=1053.298,386.128,-119.733,174.164,39.929,157.691
C06103=1053.290,385.882,-119.692,174.158,39.922,157.689
C06104=1053.282,385.635,-119.651,174.151,39.916,157.687
C06105=1053.274,385.389,-119.609,174.145,39.910,157.685
C06106=1053.266,385.143,-119.569,174.139,39.903,157.683
C06107=1053.258,384.895,-119.527,174.133,39.897,157.682
C06108=1053.250,384.650,-119.486,174.127,39.891,157.680
C06109=1053.242,384.403,-119.445,174.120,39.884,157.678
C06110=1053.234,384.157,-119.404,174.114,39.878,157.676
C06111=1053.226,383.911,-119.363,174.108,39.872,157.674
C06112=1053.219,383.664,-119.322,174.102,39.865,157.673
C06113=1053.210,383.417,-119.281,174.096,39.860,157.671
C06114=1053.202,383.171,-119.240,174.089,39.853,157.669
C06115=1053.195,382.925,-119.198,174.083,39.847,157.667
C06116=1053.187,382.679,-119.158,174.078,39.840,157.666
C06117=1053.179,382.432,-119.117,174.072,39.835,157.664
C06118=1053.172,382.186,-119.076,174.065,39.828,157.662
C06119=1053.163,381.939,-119.035,174.059,39.822,157.660
C06120=1053.156,381.692,-118.995,174.054,39.816,157.659
C06121=1053.148,381.446,-118.954,174.047,39.810,157.657
C06122=1053.140,381.200,-118.914,174.041,39.804,157.655
C06123=1053.132,380.953,-118.873,174.035,39.798,157.654
C06124=1053.125,380.707,-118.832,174.030,39.792,157.652
C06125=1053.117,380.460,-118.791,174.023,39.785,157.650
C06126=1053.109,380.214,-118.751,174.017,39.780,157.649
C06127=1053.100,379.942,-118.706,174.010,39.773,157.647
C06128=1053.092,379.670,-118.661,174.005,39.766,157.645
C06129=1053.084,379.399,-118.617,173.998,39.760,157.643
C06130=1053.074,379.128,-118.573,173.991,39.753,157.641
C06131=1053.066,378.882,-118.532,173.985,39.747,157.639
C06132=1053.059,378.635,-118.492,173.980,39.741,157.638
C06133=1053.051,378.388,-118.452,173.974,39.735,157.636
C06134=1053.043,378.141,-118.412,173.968,39.730,157.635
C06135=1053.035,377.895,-118.371,173.962,39.724,157.633
C06136=1053.028,377.649,-118.332,173.956,39.718,157.631
C06137=1053.020,377.403,-118.291,173.951,39.712,157.630
C06138=1053.012,377.156,-118.251,173.945,39.706,157.628
C06139=1053.004,376.909,-118.211,173.939,39.700,157.626
C06140=1052.996,376.663,-118.170,173.933,39.695,157.625
C06141=1052.989,376.416,-118.131,173.927,39.689,157.623
C06142=1052.981,376.169,-118.091,173.922,39.683,157.622
C06143=1052.973,375.923,-118.050,173.916,39.677,157.620
C06144=1052.966,375.676,-118.010,173.910,39.671,157.618
C06145=1052.958,375.429,-117.971,173.905,39.665,157.617
C06146=1052.950,375.182,-117.931,173.899,39.660,157.615
C06147=1052.942,374.903,-117.885,173.892,39.653,157.613
C06148=1052.933,374.624,-117.841,173.886,39.647,157.612
C06149=1052.924,374.344,-117.795,173.880,39.640,157.610
C06150=1052.916,374.065,-117.750,173.873,39.634,157.608
C06151=1052.908,373.818,-117.710,173.868,39.628,157.606
C06152=1052.901,373.572,-117.670,173.862,39.623,157.605
C06153=1052.893,373.325,-117.630,173.856,39.617,157.603
C06154=1052.886,373.078,-117.590,173.851,39.611,157.602
C06155=1052.878,372.832,-117.550,173.845,39.606,157.600
C06156=1052.871,372.585,-117.512,173.840,39.600,157.599
C06157=1052.863,372.338,-117.472,173.834,39.594,157.597
C06158=1052.855,372.091,-117.432,173.829,39.588,157.596
C06159=1052.848,371.845,-117.393,173.823,39.583,157.594
C06160=1052.840,371.598,-117.353,173.818,39.577,157.592
C06161=1052.832,371.351,-117.313,173.812,39.572,157.591
C06162=1052.825,371.105,-117.275,173.807,39.566,157.590
C06163=1052.817,370.858,-117.235,173.801,39.561,157.588
C06164=1052.810,370.610,-117.196,173.796,39.555,157.586
C06165=1052.802,370.364,-117.157,173.790,39.550,157.585
C06166=1052.794,370.117,-117.117,173.785,39.545,157.584
C06167=1052.787,369.871,-117.078,173.780,39.539,157.582
C06168=1052.779,369.624,-117.039,173.774,39.533,157.580
C06169=1052.772,369.377,-117.000,173.769,39.528,157.579
C06170=1052.764,369.131,-116.960,173.763,39.523,157.578
C06171=1052.756,368.883,-116.921,173.758,39.517,157.576
C06172=1052.749,368.637,-116.882,173.752,39.512,157.575
C06173=1052.741,368.390,-116.843,173.747,39.507,157.573
C06174=1052.734,368.143,-116.804,173.741,39.501,157.572
C06175=1052.726,367.896,-116.765,173.736,39.496,157.570
C06176=1052.719,367.649,-116.726,173.731,39.490,157.569
C06177=1052.712,367.403,-116.687,173.725,39.485,157.567
C06178=1052.704,367.156,-116.648,173.720,39.480,157.566
C06179=1052.697,366.909,-116.609,173.714,39.474,157.564
C06180=1052.688,366.663,-116.570,173.710,39.469,157.563
C06181=1052.682,366.416,-116.531,173.705,39.464,157.561
C06182=1052.673,366.169,-116.492,173.699,39.458,157.560
C06183=1052.667,365.922,-116.453,173.694,39.453,157.559
C06184=1052.660,365.675,-116.415,173.688,39.448,157.557
C06185=1052.651,365.428,-116.375,173.683,39.443,157.556
C06186=1052.645,365.181,-116.336,173.678,39.437,157.554
C06187=1052.637,364.935,-116.298,173.673,39.432,157.553
C06188=1052.630,364.687,-116.259,173.668,39.427,157.552
C06189=1052.622,364.441,-116.221,173.663,39.422,157.550
C06190=1052.615,364.194,-116.182,173.657,39.416,157.549
C06191=1052.608,363.948,-116.144,173.652,39.411,157.547
C06192=1052.600,363.700,-116.104,173.646,39.406,157.546
C06193=1052.593,363.453,-116.066,173.642,39.401,157.544
C06194=1052.586,363.207,-116.027,173.637,39.396,157.543
C06195=1052.578,362.960,-115.989,173.631,39.390,157.542
C06196=1052.571,362.713,-115.950,173.626,39.386,157.540
C06197=1052.564,362.466,-115.912,173.621,39.380,157.539
C06198=1052.556,362.219,-115.874,173.617,39.375,157.538
C06199=1052.549,361.971,-115.835,173.611,39.370,157.536
C06200=1052.541,361.725,-115.797,173.606,39.365,157.535
C06201=1052.534,361.478,-115.759,173.600,39.360,157.533
C06202=1052.526,361.231,-115.721,173.595,39.355,157.532
C06203=1052.518,360.945,-115.676,173.590,39.349,157.530
C06204=1052.510,360.661,-115.632,173.584,39.343,157.529
C06205=1052.501,360.375,-115.587,173.578,39.338,157.527
C06206=1052.492,360.090,-115.543,173.572,39.332,157.526
C06207=1052.485,359.843,-115.506,173.567,39.327,157.524
C06208=1052.478,359.596,-115.468,173.563,39.321,157.523
C06209=1052.470,359.349,-115.430,173.557,39.317,157.522
C06210=1052.463,359.101,-115.391,173.552,39.312,157.520
C06211=1052.456,358.854,-115.353,173.547,39.307,157.519
C06212=1052.448,358.608,-115.315,173.543,39.302,157.518
C06213=1052.441,358.361,-115.278,173.537,39.297,157.516
C06214=1052.433,358.114,-115.239,173.532,39.292,157.515
C06215=1052.427,357.867,-115.201,173.528,39.287,157.514
C06216=1052.420,357.619,-115.164,173.523,39.282,157.512
C06217=1052.412,357.373,-115.126,173.517,39.277,157.511
C06218=1052.405,357.126,-115.088,173.513,39.272,157.510
C06219=1052.398,356.879,-115.051,173.508,39.267,157.509
C06220=1052.390,356.632,-115.012,173.503,39.263,157.507
C06221=1052.383,356.385,-114.975,173.498,39.258,157.506
C06222=1052.376,356.138,-114.937,173.493,39.253,157.505
C06223=1052.368,355.891,-114.900,173.488,39.248,157.503
C06224=1052.361,355.644,-114.862,173.484,39.243,157.502
C06225=1052.354,355.396,-114.825,173.479,39.238,157.501
C06226=1052.346,355.150,-114.786,173.473,39.234,157.500
C06227=1052.339,354.903,-114.749,173.469,39.229,157.498
C06228=1052.332,354.656,-114.711,173.464,39.224,157.497
C06229=1052.325,354.409,-114.674,173.459,39.219,157.496
C06230=1052.317,354.161,-114.636,173.455,39.214,157.494
C06231=1052.310,353.914,-114.599,173.449,39.209,157.493
C06232=1052.303,353.667,-114.561,173.445,39.205,157.492
C06233=1052.296,353.420,-114.524,173.440,39.200,157.491
C06234=1052.288,353.173,-114.486,173.435,39.195,157.489
C06235=1052.281,352.926,-114.449,173.431,39.190,157.488
C06236=1052.274,352.679,-114.411,173.425,39.186,157.487
C06237=1052.267,352.432,-114.374,173.421,39.181,157.486
C06238=1052.260,352.184,-114.337,173.416,39.176,157.484
C06239=1052.253,351.937,-114.300,173.412,39.172,157.483
C06240=1052.246,351.690,-114.262,173.407,39.167,157.482
C06241=1052.239,351.443,-114.225,173.402,39.162,157.481
C06242=1052.231,351.196,-114.187,173.398,39.158,157.479
C06243=1052.225,350.949,-114.151,173.392,39.153,157.478
C06244=1052.217,350.702,-114.114,173.388,39.149,157.477
C06245=1052.210,350.455,-114.076,173.383,39.144,157.476
C06246=1052.203,350.207,-114.039,173.379,39.139,157.475
C06247=1052.196,349.960,-114.002,173.374,39.134,157.473
C06248=1052.188,349.713,-113.965,173.370,39.130,157.472
C06249=1052.181,349.466,-113.928,173.364,39.125,157.471
C06250=1052.174,349.219,-113.891,173.360,39.121,157.470
C06251=1052.167,348.971,-113.854,173.355,39.116,157.469
C06252=1052.159,348.724,-113.817,173.351,39.111,157.467
C06253=1052.153,348.477,-113.781,173.346,39.107,157.466
C06254=1052.146,348.230,-113.743,173.342,39.103,157.465
C06255=1052.139,347.982,-113.706,173.337,39.098,157.464
C06256=1052.131,347.736,-113.669,173.333,39.093,157.463
C06257=1052.124,347.489,-113.633,173.328,39.089,157.461
C06258=1052.117,347.241,-113.595,173.323,39.084,157.460
C06259=1052.109,346.961,-113.555,173.318,39.079,157.459
C06260=1052.100,346.681,-113.512,173.313,39.074,157.457
C06261=1052.093,346.400,-113.471,173.308,39.069,157.456
C06262=1052.085,346.120,-113.430,173.303,39.064,157.455
C06263=1052.078,345.873,-113.392,173.299,39.060,157.454
C06264=1052.071,345.626,-113.356,173.293,39.055,157.452
C06265=1052.064,345.379,-113.319,173.289,39.050,157.451
C06266=1052.057,345.131,-113.283,173.284,39.046,157.450
C06267=1052.049,344.885,-113.246,173.280,39.042,157.449
C06268=1052.042,344.637,-113.209,173.275,39.037,157.448
C06269=1052.035,344.390,-113.173,173.271,39.033,157.447
C06270=1052.028,344.142,-113.137,173.267,39.028,157.446
C06271=1052.022,343.895,-113.100,173.262,39.024,157.444
C06272=1052.014,343.648,-113.064,173.258,39.020,157.443
C06273=1052.008,343.400,-113.027,173.253,39.015,157.442
C06274=1052.000,343.154,-112.991,173.249,39.010,157.441
C06275=1051.993,342.906,-112.954,173.245,39.006,157.440
C06276=1051.986,342.660,-112.918,173.240,39.002,157.439
C06277=1051.979,342.412,-112.881,173.236,38.998,157.438
C06278=1051.972,342.164,-112.846,173.232,38.993,157.436
C06279=1051.965,341.917,-112.809,173.227,38.989,157.435
C06280=1051.958,341.670,-112.773,173.223,38.985,157.434
C06281=1051.951,341.423,-112.737,173.218,38.980,157.433
C06282=1051.944,341.175,-112.701,173.213,38.976,157.432
C06283=1051.937,340.928,-112.664,173.209,38.972,157.431
C06284=1051.930,340.681,-112.629,173.204,38.967,157.430
C06285=1051.923,340.434,-112.592,173.200,38.963,157.429
C06286=1051.916,340.186,-112.557,173.196,38.959,157.428
C06287=1051.908,339.939,-112.520,173.191,38.955,157.426
C06288=1051.902,339.692,-112.484,173.187,38.950,157.425
C06289=1051.895,339.445,-112.448,173.183,38.946,157.424
C06290=1051.887,339.197,-112.413,173.178,38.942,157.423
C06291=1051.881,338.950,-112.376,173.174,38.938,157.422
C06292=1051.873,338.702,-112.340,173.170,38.933,157.421
C06293=1051.867,338.455,-112.305,173.165,38.929,157.420
C06294=1051.860,338.208,-112.268,173.161,38.925,157.419
C06295=1051.853,337.961,-112.232,173.157,38.920,157.418
C06296=1051.846,337.713,-112.197,173.153,38.916,157.416
C06297=1051.840,337.466,-112.161,173.148,38.912,157.415
C06298=1051.832,337.218,-112.125,173.144,38.908,157.414
C06299=1051.825,336.971,-112.089,173.140,38.903,157.413
C06300=1051.819,336.724,-112.053,173.136,38.900,157.412
C06301=1051.811,336.476,-112.017,173.131,38.895,157.411
C06302=1051.805,336.229,-111.982,173.128,38.891,157.410
C06303=1051.798,335.982,-111.946,173.124,38.887,157.409
C06304=1051.790,335.734,-111.911,173.119,38.883,157.408
C06305=1051.784,335.487,-111.874,173.115,38.879,157.407
C06306=1051.777,335.240,-111.839,173.111,38.875,157.406
C06307=1051.770,334.991,-111.804,173.107,38.870,157.405
C06308=1051.763,334.745,-111.768,173.102,38.867,157.404
C06309=1051.756,334.497,-111.733,173.098,38.862,157.403
C06310=1051.749,334.250,-111.698,173.094,38.858,157.402
C06311=1051.741,334.003,-111.661,173.090,38.854,157.400
C06312=1051.735,333.755,-111.626,173.086,38.850,157.399
C06313=1051.728,333.508,-111.591,173.081,38.846,157.398
C06314=1051.721,333.260,-111.556,173.077,38.842,157.397
C06315=1051.713,332.976,-111.515,173.072,38.837,157.396
C06316=1051.705,332.692,-111.474,173.068,38.832,157.395
C06317=1051.697,332.408,-111.434,173.063,38.828,157.394
C06318=1051.690,332.123,-111.393,173.058,38.823,157.393
C06319=1051.683,331.876,-111.357,173.054,38.819,157.392
C06320=1051.676,331.628,-111.322,173.050,38.815,157.390
C06321=1051.669,331.381,-111.287,173.046,38.811,157.389
C06322=1051.662,331.133,-111.252,173.042,38.807,157.388
C06323=1051.655,330.886,-111.217,173.038,38.803,157.388
C06324=1051.649,330.639,-111.181,173.033,38.799,157.386
C06325=1051.642,330.391,-111.146,173.029,38.795,157.385
C06326=1051.635,330.144,-111.111,173.025,38.791,157.384
C06327=1051.628,329.896,-111.076,173.021,38.787,157.383
C06328=1051.622,329.649,-111.041,173.018,38.783,157.382
C06329=1051.613,329.401,-111.006,173.014,38.779,157.381
C06330=1051.607,329.154,-110.971,173.010,38.775,157.380
C06331=1051.600,328.907,-110.936,173.005,38.771,157.379
C06332=1051.593,328.659,-110.902,173.001,38.767,157.378
C06333=1051.586,328.412,-110.867,172.997,38.763,157.377
C06334=1051.579,328.164,-110.832,172.993,38.759,157.376
C06335=1051.572,327.917,-110.797,172.989,38.756,157.375
C06336=1051.564,327.669,-110.762,172.986,38.752,157.374
C06337=1051.558,327.421,-110.727,172.981,38.748,157.373
C06338=1051.550,327.174,-110.693,172.977,38.744,157.372
C06339=1051.544,326.927,-110.657,172.973,38.740,157.371
C06340=1051.536,326.679,-110.624,172.969,38.736,157.370
C06341=1051.530,326.432,-110.588,172.965,38.732,157.370
C06342=1051.523,326.184,-110.553,172.961,38.728,157.369
C06343=1051.516,325.937,-110.520,172.957,38.725,157.368
C06344=1051.509,325.689,-110.484,172.954,38.721,157.367
C06345=1051.502,325.441,-110.450,172.950,38.717,157.366
C06346=1051.495,325.194,-110.415,172.946,38.713,157.365
C06347=1051.488,324.947,-110.380,172.941,38.709,157.364
C06348=1051.481,324.699,-110.346,172.937,38.705,157.363
C06349=1051.474,324.452,-110.311,172.933,38.702,157.362
C06350=1051.468,324.204,-110.277,172.930,38.698,157.361
C06351=1051.460,323.957,-110.242,172.926,38.694,157.360
C06352=1051.454,323.709,-110.208,172.922,38.690,157.359
C06353=1051.446,323.461,-110.174,172.918,38.686,157.358
C06354=1051.440,323.214,-110.139,172.914,38.682,157.357
C06355=1051.434,322.966,-110.105,172.910,38.679,157.356
C06356=1051.426,322.719,-110.070,172.906,38.675,157.355
C06357=1051.420,322.471,-110.036,172.903,38.671,157.354
C06358=1051.412,322.224,-110.001,172.899,38.667,157.353
C06359=1051.406,321.976,-109.967,172.895,38.664,157.352
C06360=1051.399,321.728,-109.933,172.891,38.660,157.351
C06361=1051.392,321.481,-109.898,172.887,38.656,157.350
C06362=1051.386,321.234,-109.864,172.883,38.652,157.349
C06363=1051.379,320.986,-109.830,172.880,38.649,157.348
C06364=1051.372,320.738,-109.796,172.876,38.645,157.347
C06365=1051.365,320.491,-109.761,172.872,38.641,157.346
C06366=1051.358,320.243,-109.727,172.868,38.637,157.345
C06367=1051.352,319.996,-109.693,172.864,38.634,157.345
C06368=1051.345,319.748,-109.659,172.860,38.630,157.344
C06369=1051.339,319.501,-109.624,172.857,38.626,157.343
C06370=1051.331,319.253,-109.590,172.853,38.622,157.342
C06371=1051.324,318.964,-109.551,172.849,38.617,157.341
C06372=1051.317,318.674,-109.511,172.844,38.613,157.340
C06373=1051.308,318.385,-109.470,172.840,38.609,157.339
C06374=1051.300,318.096,-109.431,172.835,38.605,157.337
C06375=1051.294,317.848,-109.397,172.831,38.601,157.336
C06376=1051.288,317.600,-109.362,172.827,38.597,157.336
C06377=1051.281,317.353,-109.329,172.824,38.593,157.335
C06378=1051.274,317.105,-109.294,172.821,38.589,157.334
C06379=1051.268,316.858,-109.261,172.817,38.585,157.333
C06380=1051.261,316.610,-109.226,172.813,38.582,157.332
C06381=1051.254,316.362,-109.193,172.809,38.578,157.331
C06382=1051.248,316.115,-109.158,172.805,38.574,157.330
C06383=1051.241,315.867,-109.125,172.802,38.571,157.329
C06384=1051.235,315.620,-109.091,172.798,38.567,157.328
C06385=1051.228,315.372,-109.057,172.794,38.564,157.327
C06386=1051.221,315.124,-109.022,172.790,38.560,157.326
C06387=1051.215,314.877,-108.989,172.786,38.556,157.325
C06388=1051.208,314.629,-108.954,172.784,38.553,157.324
C06389=1051.202,314.382,-108.921,172.780,38.549,157.324
C06390=1051.194,314.135,-108.887,172.776,38.545,157.323
C06391=1051.189,313.887,-108.854,172.772,38.541,157.322
C06392=1051.182,313.639,-108.820,172.768,38.537,157.321
C06393=1051.176,313.392,-108.786,172.765,38.534,157.320
C06394=1051.169,313.144,-108.752,172.761,38.530,157.319
C06395=1051.162,312.895,-108.718,172.757,38.527,157.318
C06396=1051.155,312.649,-108.686,172.754,38.523,157.317
C06397=1051.148,312.401,-108.652,172.751,38.519,157.316
C06398=1051.142,312.154,-108.619,172.747,38.516,157.315
C06399=1051.134,311.906,-108.585,172.743,38.512,157.315
C06400=1051.128,311.658,-108.552,172.739,38.509,157.314
C06401=1051.121,311.411,-108.519,172.736,38.506,157.313
C06402=1051.114,311.162,-108.486,172.732,38.502,157.312
C06403=1051.107,310.915,-108.452,172.728,38.498,157.311
C06404=1051.100,310.668,-108.418,172.724,38.495,157.310
C06405=1051.093,310.419,-108.385,172.722,38.491,157.309
C06406=1051.087,310.172,-108.352,172.718,38.488,157.308
C06407=1051.080,309.924,-108.319,172.714,38.484,157.308
C06408=1051.074,309.677,-108.286,172.710,38.481,157.307
C06409=1051.066,309.429,-108.252,172.707,38.478,157.306
C06410=1051.060,309.181,-108.219,172.703,38.474,157.305
C06411=1051.052,308.934,-108.186,172.700,38.470,157.304
C06412=1051.046,308.686,-108.153,172.696,38.467,157.303
C06413=1051.039,308.438,-108.120,172.693,38.463,157.302
C06414=1051.032,308.191,-108.087,172.689,38.460,157.302
C06415=1051.026,307.943,-108.054,172.685,38.456,157.301
C06416=1051.019,307.695,-108.021,172.682,38.453,157.300
C06417=1051.013,307.448,-107.987,172.679,38.449,157.299
C06418=1051.006,307.200,-107.954,172.675,38.446,157.298
C06419=1050.999,306.952,-107.922,172.671,38.442,157.297
C06420=1050.992,306.705,-107.888,172.668,38.439,157.296
C06421=1050.985,306.457,-107.856,172.664,38.435,157.296
C06422=1050.979,306.210,-107.823,172.661,38.432,157.295
C06423=1050.972,305.961,-107.790,172.657,38.429,157.294
C06424=1050.965,305.714,-107.756,172.654,38.425,157.293
C06425=1050.959,305.467,-107.724,172.650,38.421,157.292
C06426=1050.952,305.219,-107.690,172.646,38.418,157.291
C06427=1050.945,304.934,-107.652,172.642,38.414,157.290
C06428=1050.936,304.648,-107.615,172.639,38.410,157.289
C06429=1050.929,304.364,-107.577,172.635,38.406,157.288
C06430=1050.922,304.079,-107.540,172.631,38.402,157.287
C06431=1050.915,303.831,-107.507,172.627,38.399,157.287
C06432=1050.908,303.583,-107.474,172.623,38.395,157.286
C06433=1050.902,303.335,-107.441,172.621,38.391,157.285
C06434=1050.896,303.088,-107.408,172.617,38.388,157.284
C06435=1050.888,302.840,-107.376,172.613,38.385,157.283
C06436=1050.882,302.593,-107.342,172.610,38.381,157.282
C06437=1050.875,302.345,-107.310,172.607,38.378,157.282
C06438=1050.869,302.097,-107.277,172.603,38.375,157.281
C06439=1050.863,301.849,-107.245,172.600,38.371,157.280
C06440=1050.856,301.601,-107.212,172.597,38.368,157.279
C06441=1050.849,301.354,-107.180,172.593,38.364,157.278
C06442=1050.843,301.106,-107.147,172.589,38.360,157.277
C06443=1050.836,300.858,-107.114,172.586,38.357,157.277
C06444=1050.830,300.610,-107.081,172.583,38.354,157.276
C06445=1050.823,300.363,-107.048,172.579,38.350,157.275
C06446=1050.816,300.115,-107.016,172.576,38.347,157.274
C06447=1050.810,299.868,-106.983,172.573,38.343,157.273
C06448=1050.804,299.620,-106.951,172.569,38.340,157.272
C06449=1050.798,299.372,-106.919,172.566,38.337,157.272
C06450=1050.791,299.124,-106.886,172.563,38.333,157.271
C06451=1050.784,298.876,-106.853,172.559,38.330,157.270
C06452=1050.777,298.629,-106.821,172.555,38.327,157.269
C06453=1050.771,298.381,-106.788,172.553,38.323,157.268
C06454=1050.765,298.133,-106.756,172.549,38.319,157.267
C06455=1050.759,297.885,-106.723,172.546,38.316,157.267
C06456=1050.752,297.638,-106.691,172.543,38.312,157.266
C06457=1050.746,297.390,-106.659,172.539,38.309,157.265
C06458=1050.740,297.142,-106.626,172.536,38.306,157.264
C06459=1050.733,296.895,-106.593,172.533,38.302,157.263
C06460=1050.727,296.646,-106.561,172.529,38.299,157.262
C06461=1050.720,296.398,-106.529,172.526,38.295,157.262
C06462=1050.713,296.151,-106.496,172.522,38.292,157.261
C06463=1050.707,295.903,-106.465,172.520,38.289,157.260
C06464=1050.700,295.655,-106.432,172.516,38.285,157.259
C06465=1050.694,295.407,-106.400,172.512,38.282,157.258
C06466=1050.687,295.160,-106.368,172.510,38.279,157.258
C06467=1050.681,294.912,-106.336,172.506,38.276,157.257
C06468=1050.674,294.664,-106.304,172.503,38.272,157.256
C06469=1050.668,294.416,-106.272,172.500,38.269,157.255
C06470=1050.661,294.169,-106.239,172.496,38.265,157.254
C06471=1050.655,293.921,-106.208,172.493,38.262,157.254
C06472=1050.648,293.673,-106.175,172.490,38.258,157.253
C06473=1050.641,293.425,-106.143,172.486,38.256,157.252
C06474=1050.634,293.177,-106.112,172.484,38.252,157.251
C06475=1050.628,292.929,-106.079,172.480,38.249,157.250
C06476=1050.621,292.681,-106.048,172.477,38.245,157.250
C06477=1050.615,292.433,-106.016,172.473,38.242,157.249
C06478=1050.608,292.186,-105.984,172.471,38.239,157.248
C06479=1050.601,291.938,-105.952,172.467,38.236,157.247
C06480=1050.595,291.690,-105.921,172.464,38.232,157.247
C06481=1050.589,291.442,-105.889,172.461,38.229,157.246
C06482=1050.582,291.195,-105.857,172.457,38.226,157.245
C06483=1050.575,290.926,-105.822,172.455,38.222,157.244
C06484=1050.568,290.656,-105.787,172.451,38.219,157.243
C06485=1050.561,290.387,-105.753,172.447,38.215,157.242
C06486=1050.554,290.119,-105.719,172.444,38.212,157.242
C06487=1050.547,289.871,-105.687,172.441,38.208,157.241
C06488=1050.541,289.623,-105.655,172.437,38.205,157.240
C06489=1050.534,289.375,-105.624,172.435,38.202,157.239
C06490=1050.528,289.127,-105.593,172.431,38.199,157.239
C06491=1050.521,288.879,-105.561,172.428,38.195,157.238
C06492=1050.515,288.631,-105.528,172.425,38.192,157.237
C06493=1050.508,288.383,-105.497,172.421,38.189,157.236
C06494=1050.501,288.135,-105.465,172.418,38.186,157.235
C06495=1050.494,287.888,-105.434,172.415,38.182,157.235
C06496=1050.488,287.640,-105.403,172.412,38.179,157.234
C06497=1050.482,287.391,-105.371,172.408,38.176,157.233
C06498=1050.475,287.144,-105.339,172.406,38.173,157.232
C06499=1050.468,286.896,-105.308,172.402,38.169,157.231
C06500=1050.462,286.648,-105.277,172.400,38.166,157.231
C06501=1050.455,286.401,-105.245,172.396,38.163,157.230
C06502=1050.449,286.152,-105.214,172.393,38.160,157.229
C06503=1050.442,285.904,-105.183,172.390,38.157,157.228
C06504=1050.436,285.656,-105.152,172.387,38.153,157.228
C06505=1050.429,285.408,-105.120,172.383,38.150,157.227
C06506=1050.422,285.160,-105.089,172.381,38.147,157.226
C06507=1050.415,284.912,-105.057,172.377,38.143,157.225
C06508=1050.409,284.665,-105.026,172.375,38.141,157.225
C06509=1050.403,284.417,-104.996,172.371,38.137,157.224
C06510=1050.396,284.169,-104.964,172.368,38.134,157.223
C06511=1050.389,283.921,-104.933,172.365,38.131,157.222
C06512=1050.383,283.673,-104.901,172.362,38.127,157.222
C06513=1050.376,283.425,-104.870,172.360,38.125,157.221
C06514=1050.370,283.177,-104.839,172.356,38.121,157.220
C06515=1050.363,282.929,-104.808,172.353,38.118,157.219
C06516=1050.357,282.682,-104.777,172.350,38.115,157.219
C06517=1050.350,282.433,-104.746,172.347,38.111,157.218
C06518=1050.344,282.185,-104.714,172.343,38.109,157.217
C06519=1050.338,281.937,-104.682,172.341,38.105,157.216
C06520=1050.332,281.689,-104.652,172.337,38.102,157.216
C06521=1050.325,281.441,-104.621,172.335,38.099,157.215
C06522=1050.318,281.193,-104.589,172.332,38.095,157.214
C06523=1050.312,280.945,-104.558,172.328,38.093,157.213
C06524=1050.306,280.698,-104.527,172.326,38.089,157.213
C06525=1050.299,280.450,-104.496,172.322,38.086,157.212
C06526=1050.293,280.201,-104.465,172.320,38.083,157.211
C06527=1050.287,279.954,-104.434,172.317,38.079,157.210
C06528=1050.280,279.705,-104.403,172.313,38.077,157.210
C06529=1050.273,279.457,-104.372,172.311,38.073,157.209
C06530=1050.266,279.209,-104.342,172.307,38.070,157.208
C06531=1050.260,278.962,-104.311,172.304,38.067,157.207
C06532=1050.254,278.714,-104.280,172.302,38.064,157.207
C06533=1050.247,278.466,-104.249,172.298,38.060,157.206
C06534=1050.241,278.217,-104.218,172.296,38.058,157.205
C06535=1050.234,277.970,-104.188,172.292,38.054,157.204
C06536=1050.227,277.722,-104.157,172.290,38.051,157.204
C06537=1050.221,277.473,-104.126,172.287,38.048,157.203
C06538=1050.215,277.226,-104.095,172.283,38.045,157.202
C06539=1050.207,276.968,-104.063,172.281,38.042,157.201
C06540=1050.200,276.710,-104.032,172.277,38.039,157.201
C06541=1050.194,276.452,-104.000,172.274,38.035,157.200
C06542=1050.187,276.195,-103.967,172.271,38.032,157.199
C06543=1050.181,275.947,-103.937,172.268,38.029,157.198
C06544=1050.174,275.699,-103.907,172.266,38.025,157.198
C06545=1050.167,275.451,-103.875,172.262,38.023,157.197
C06546=1050.162,275.203,-103.845,172.259,38.019,157.196
C06547=1050.155,274.955,-103.814,172.257,38.016,157.196
C06548=1050.148,274.707,-103.784,172.253,38.013,157.195
C06549=1050.142,274.459,-103.754,172.251,38.010,157.194
C06550=1050.135,274.211,-103.723,172.248,38.007,157.193
C06551=1050.129,273.963,-103.693,172.245,38.004,157.193
C06552=1050.123,273.715,-103.662,172.242,38.001,157.192
C06553=1050.116,273.466,-103.631,172.239,37.997,157.191
C06554=1050.110,273.219,-103.602,172.236,37.994,157.190
C06555=1050.103,272.970,-103.571,172.233,37.991,157.190
C06556=1050.097,272.723,-103.540,172.231,37.988,157.189
C06557=1050.090,272.475,-103.510,172.227,37.985,157.188
C06558=1050.083,272.226,-103.479,172.225,37.982,157.188
C06559=1050.078,271.979,-103.449,172.222,37.979,157.187
C06560=1050.070,271.730,-103.418,172.218,37.975,157.186
C06561=1050.065,271.483,-103.388,172.216,37.973,157.185
C06562=1050.057,271.234,-103.358,172.213,37.969,157.185
C06563=1050.051,270.986,-103.327,172.211,37.966,157.184
C06564=1050.044,270.738,-103.298,172.207,37.963,157.183
C06565=1050.038,270.490,-103.267,172.204,37.960,157.182
C06566=1050.032,270.242,-103.237,172.202,37.957,157.182
C06567=1050.025,269.994,-103.206,172.198,37.954,157.181
C06568=1050.019,269.746,-103.177,172.196,37.951,157.180
C06569=1050.012,269.498,-103.146,172.193,37.948,157.180
C06570=1050.006,269.250,-103.116,172.191,37.944,157.179
C06571=1049.999,269.002,-103.085,172.187,37.941,157.178
C06572=1049.993,268.754,-103.056,172.185,37.938,157.178
C06573=1049.986,268.505,-103.026,172.182,37.935,157.177
C06574=1049.980,268.258,-102.996,172.178,37.932,157.176
C06575=1049.974,268.009,-102.965,172.176,37.929,157.175
C06576=1049.967,267.761,-102.935,172.173,37.926,157.175
C06577=1049.961,267.513,-102.905,172.171,37.923,157.174
C06578=1049.954,267.265,-102.876,172.167,37.920,157.173
C06579=1049.947,267.017,-102.846,172.165,37.917,157.172
C06580=1049.941,266.769,-102.815,172.162,37.914,157.172
C06581=1049.934,266.521,-102.785,172.159,37.911,157.171
C06582=1049.928,266.272,-102.756,172.156,37.907,157.170
C06583=1049.921,266.024,-102.725,172.153,37.904,157.170
C06584=1049.915,265.776,-102.696,172.151,37.901,157.169
C06585=1049.908,265.528,-102.666,172.148,37.898,157.168
C06586=1049.902,265.280,-102.636,172.146,37.895,157.168
C06587=1049.896,265.032,-102.606,172.142,37.892,157.167
C06588=1049.889,264.783,-102.577,172.140,37.889,157.166
C06589=1049.883,264.536,-102.546,172.137,37.886,157.165
C06590=1049.876,264.287,-102.516,172.134,37.883,157.165
C06591=1049.870,264.039,-102.487,172.131,37.880,157.164
C06592=1049.864,263.791,-102.457,172.128,37.877,157.163
C06593=1049.857,263.543,-102.427,172.126,37.874,157.163
C06594=1049.850,263.295,-102.398,172.123,37.871,157.162
C06595=1049.844,263.041,-102.366,172.121,37.867,157.161
C06596=1049.837,262.788,-102.336,172.117,37.864,157.161
C06597=1049.831,262.535,-102.306,172.115,37.861,157.160
C06598=1049.824,262.281,-102.276,172.112,37.858,157.159
C06599=1049.817,262.034,-102.246,172.109,37.855,157.158
C06600=1049.811,261.785,-102.217,172.107,37.852,157.158
C06601=1049.804,261.537,-102.188,172.103,37.849,157.157
C06602=1049.798,261.289,-102.158,172.101,37.846,157.156
C06603=1049.791,261.040,-102.129,172.098,37.843,157.156
C06604=1049.784,260.793,-102.099,172.096,37.840,157.155
C06605=1049.778,260.544,-102.069,172.093,37.837,157.154
C06606=1049.771,260.296,-102.040,172.090,37.834,157.154
C06607=1049.765,260.048,-102.011,172.087,37.831,157.153
C06608=1049.757,259.800,-101.982,172.085,37.828,157.152
C06609=1049.751,259.552,-101.953,172.082,37.825,157.152
C06610=1049.744,259.304,-101.923,172.080,37.822,157.151
C06611=1049.738,259.055,-101.894,172.076,37.819,157.150
C06612=1049.731,258.807,-101.865,172.074,37.816,157.150
C06613=1049.724,258.559,-101.834,172.071,37.813,157.149
C06614=1049.718,258.311,-101.805,172.068,37.810,157.148
C06615=1049.712,258.063,-101.776,172.066,37.807,157.147
C06616=1049.705,257.814,-101.747,172.063,37.804,157.147
C06617=1049.699,257.566,-101.718,172.061,37.801,157.146
C06618=1049.692,257.318,-101.688,172.057,37.798,157.145
C06619=1049.685,257.070,-101.659,172.055,37.795,157.145
C06620=1049.679,256.821,-101.630,172.052,37.792,157.144
C06621=1049.673,256.573,-101.601,172.050,37.789,157.143
C06622=1049.666,256.325,-101.572,172.047,37.786,157.143
C06623=1049.659,256.077,-101.541,172.045,37.783,157.142
C06624=1049.653,255.829,-101.512,172.042,37.780,157.141
C06625=1049.647,255.581,-101.483,172.040,37.777,157.141
C06626=1049.640,255.332,-101.454,172.036,37.774,157.140
C06627=1049.633,255.084,-101.426,172.034,37.771,157.139
C06628=1049.627,254.836,-101.397,172.031,37.768,157.139
C06629=1049.620,254.588,-101.367,172.028,37.764,157.138
C06630=1049.614,254.339,-101.338,172.026,37.762,157.137
C06631=1049.607,254.091,-101.309,172.023,37.759,157.136
C06632=1049.601,253.843,-101.280,172.021,37.756,157.136
C06633=1049.595,253.595,-101.251,172.018,37.753,157.135
C06634=1049.589,253.346,-101.222,172.016,37.749,157.134
C06635=1049.582,253.098,-101.192,172.013,37.746,157.134
C06636=1049.575,252.849,-101.163,172.011,37.743,157.133
C06637=1049.569,252.601,-101.134,172.008,37.741,157.132
C06638=1049.562,252.353,-101.106,172.005,37.737,157.132
C06639=1049.556,252.105,-101.077,172.002,37.734,157.131
C06640=1049.550,251.857,-101.048,172.000,37.731,157.130
C06641=1049.543,251.608,-101.018,171.997,37.728,157.130
C06642=1049.537,251.360,-100.989,171.995,37.725,157.129
C06643=1049.530,251.112,-100.960,171.992,37.722,157.128
C06644=1049.524,250.864,-100.931,171.990,37.719,157.128
C06645=1049.518,250.616,-100.902,171.987,37.716,157.127
C06646=1049.512,250.368,-100.873,171.985,37.713,157.126
C06647=1049.505,250.120,-100.845,171.982,37.710,157.125
C06648=1049.498,249.872,-100.816,171.979,37.707,157.125
C06649=1049.492,249.622,-100.787,171.977,37.704,157.124
C06650=1049.486,249.374,-100.758,171.974,37.701,157.123
C06651=1049.479,249.119,-100.729,171.972,37.697,157.123
C06652=1049.473,248.865,-100.698,171.969,37.694,157.122
C06653=1049.466,248.610,-100.669,171.967,37.691,157.121
C06654=1049.460,248.355,-100.640,171.964,37.688,157.121
C06655=1049.454,248.107,-100.611,171.962,37.685,157.120
C06656=1049.447,247.859,-100.582,171.959,37.682,157.119
C06657=1049.441,247.609,-100.553,171.957,37.679,157.119
C06658=1049.435,247.361,-100.524,171.954,37.676,157.118
C06659=1049.428,247.113,-100.495,171.952,37.673,157.117
C06660=1049.421,246.865,-100.467,171.949,37.669,157.116
C06661=1049.415,246.617,-100.438,171.947,37.666,157.116
C06662=1049.409,246.368,-100.409,171.944,37.663,157.115
C06663=1049.403,246.120,-100.380,171.941,37.660,157.114
C06664=1049.397,245.872,-100.352,171.939,37.657,157.114
C06665=1049.391,245.623,-100.323,171.937,37.654,157.113
C06666=1049.384,245.376,-100.294,171.934,37.651,157.112
C06667=1049.378,245.127,-100.266,171.932,37.648,157.112
C06668=1049.371,244.879,-100.238,171.929,37.645,157.111
C06669=1049.365,244.630,-100.209,171.926,37.642,157.110
C06670=1049.359,244.382,-100.180,171.924,37.639,157.110
C06671=1049.352,244.134,-100.153,171.921,37.636,157.109
C06672=1049.346,243.886,-100.124,171.919,37.633,157.108
C06673=1049.339,243.638,-100.095,171.916,37.629,157.108
C06674=1049.333,243.389,-100.067,171.914,37.626,157.107
C06675=1049.326,243.141,-100.038,171.911,37.624,157.106
C06676=1049.320,242.892,-100.010,171.909,37.621,157.106
C06677=1049.314,242.644,-99.981,171.906,37.618,157.105
C06678=1049.307,242.396,-99.953,171.905,37.614,157.104
C06679=1049.301,242.147,-99.925,171.902,37.611,157.104
C06680=1049.295,241.899,-99.896,171.900,37.608,157.103
C06681=1049.288,241.651,-99.868,171.897,37.605,157.102
C06682=1049.282,241.402,-99.839,171.895,37.602,157.102
C06683=1049.275,241.154,-99.811,171.892,37.599,157.101
C06684=1049.268,240.906,-99.784,171.890,37.596,157.100
C06685=1049.262,240.657,-99.755,171.887,37.593,157.099
C06686=1049.255,240.409,-99.727,171.885,37.590,157.099
C06687=1049.249,240.161,-99.699,171.882,37.587,157.098
C06688=1049.243,239.912,-99.670,171.880,37.584,157.098
C06689=1049.236,239.664,-99.642,171.877,37.581,157.097
C06690=1049.230,239.415,-99.614,171.875,37.578,157.096
C06691=1049.224,239.168,-99.586,171.872,37.575,157.095
C06692=1049.217,238.920,-99.558,171.871,37.572,157.095
C06693=1049.211,238.671,-99.530,171.868,37.569,157.094
C06694=1049.204,238.422,-99.502,171.866,37.566,157.093
C06695=1049.198,238.174,-99.474,171.863,37.563,157.093
C06696=1049.191,237.926,-99.445,171.861,37.560,157.092
C06697=1049.185,237.677,-99.418,171.858,37.557,157.092
C06698=1049.178,237.429,-99.390,171.856,37.554,157.091
C06699=1049.171,237.181,-99.362,171.853,37.551,157.090
C06700=1049.165,236.932,-99.334,171.851,37.548,157.089
C06701=1049.158,236.684,-99.305,171.848,37.545,157.089
C06702=1049.152,236.436,-99.278,171.847,37.542,157.088
C06703=1049.146,236.187,-99.249,171.844,37.539,157.088
C06704=1049.140,235.939,-99.222,171.842,37.536,157.087
C06705=1049.133,235.691,-99.194,171.839,37.532,157.086
C06706=1049.126,235.442,-99.167,171.837,37.529,157.085
C06707=1049.120,235.182,-99.137,171.834,37.526,157.085
C06708=1049.113,234.920,-99.107,171.832,37.523,157.084
C06709=1049.107,234.660,-99.078,171.829,37.520,157.083
C06710=1049.099,234.399,-99.049,171.827,37.517,157.083
C06711=1049.093,234.151,-99.021,171.824,37.513,157.082
C06712=1049.087,233.903,-98.993,171.823,37.511,157.081
C06713=1049.080,233.654,-98.966,171.820,37.508,157.081
C06714=1049.074,233.405,-98.937,171.818,37.505,157.080
C06715=1049.067,233.157,-98.910,171.815,37.502,157.079
C06716=1049.061,232.909,-98.882,171.813,37.498,157.079
C06717=1049.055,232.661,-98.854,171.810,37.495,157.078
C06718=1049.048,232.412,-98.827,171.809,37.492,157.077
C06719=1049.042,232.164,-98.798,171.806,37.489,157.077
C06720=1049.035,231.915,-98.771,171.804,37.486,157.076
C06721=1049.030,231.667,-98.744,171.801,37.483,157.075
C06722=1049.023,231.418,-98.716,171.799,37.480,157.075
C06723=1049.016,231.170,-98.689,171.797,37.477,157.074
C06724=1049.010,230.921,-98.661,171.795,37.474,157.073
C06725=1049.003,230.673,-98.633,171.792,37.471,157.073
C06726=1048.997,230.425,-98.606,171.790,37.468,157.072
C06727=1048.991,230.177,-98.577,171.787,37.464,157.071
C06728=1048.984,229.927,-98.550,171.786,37.461,157.071
C06729=1048.978,229.679,-98.523,171.783,37.459,157.070
C06730=1048.972,229.431,-98.495,171.781,37.456,157.069
C06731=1048.965,229.183,-98.468,171.778,37.453,157.069
C06732=1048.958,228.934,-98.440,171.776,37.449,157.068
C06733=1048.952,228.685,-98.413,171.774,37.446,157.067
C06734=1048.946,228.438,-98.385,171.772,37.443,157.067
C06735=1048.939,228.189,-98.358,171.770,37.440,157.066
C06736=1048.933,227.941,-98.330,171.767,37.437,157.065
C06737=1048.926,227.692,-98.303,171.765,37.434,157.065
C06738=1048.919,227.444,-98.276,171.763,37.431,157.064
C06739=1048.913,227.196,-98.248,171.761,37.428,157.063
C06740=1048.906,226.947,-98.221,171.758,37.425,157.063
C06741=1048.900,226.698,-98.194,171.756,37.422,157.062
C06742=1048.894,226.451,-98.166,171.753,37.419,157.061
C06743=1048.887,226.201,-98.139,171.752,37.416,157.061
C06744=1048.880,225.953,-98.112,171.749,37.413,157.060
C06745=1048.874,225.704,-98.085,171.747,37.410,157.059
C06746=1048.868,225.456,-98.057,171.744,37.407,157.059
C06747=1048.861,225.208,-98.030,171.743,37.404,157.058
C06748=1048.854,224.959,-98.003,171.740,37.401,157.057
C06749=1048.848,224.711,-97.976,171.738,37.398,157.057
C06750=1048.842,224.462,-97.949,171.735,37.395,157.056
C06751=1048.835,224.214,-97.921,171.734,37.392,157.055
C06752=1048.829,223.965,-97.894,171.731,37.389,157.055
C06753=1048.823,223.717,-97.867,171.729,37.385,157.054
C06754=1048.816,223.468,-97.840,171.727,37.382,157.053
C06755=1048.809,223.221,-97.813,171.725,37.379,157.053
C06756=1048.803,222.971,-97.786,171.722,37.376,157.052
C06757=1048.796,222.723,-97.758,171.720,37.373,157.051
C06758=1048.791,222.475,-97.731,171.718,37.370,157.051
C06759=1048.784,222.226,-97.704,171.716,37.367,157.050
C06760=1048.778,221.978,-97.677,171.714,37.364,157.049
C06761=1048.771,221.730,-97.650,171.712,37.361,157.049
C06762=1048.764,221.481,-97.623,171.710,37.358,157.048
C06763=1048.758,221.213,-97.594,171.707,37.354,157.047
C06764=1048.751,220.945,-97.564,171.704,37.351,157.047
C06765=1048.744,220.676,-97.535,171.702,37.348,157.046
C06766=1048.737,220.408,-97.506,171.700,37.344,157.045
C06767=1048.731,220.159,-97.479,171.698,37.341,157.045
C06768=1048.724,219.911,-97.453,171.696,37.338,157.044
C06769=1048.717,219.662,-97.425,171.693,37.335,157.043
C06770=1048.711,219.414,-97.398,171.692,37.332,157.042
C06771=1048.704,219.165,-97.372,171.689,37.329,157.042
C06772=1048.698,218.917,-97.345,171.687,37.326,157.041
C06773=1048.691,218.669,-97.318,171.685,37.323,157.041
C06774=1048.685,218.420,-97.291,171.683,37.320,157.040
C06775=1048.679,218.171,-97.265,171.680,37.317,157.039
C06776=1048.672,217.923,-97.237,171.679,37.314,157.039
C06777=1048.666,217.675,-97.211,171.676,37.310,157.038
C06778=1048.659,217.426,-97.184,171.674,37.307,157.037
C06779=1048.652,217.177,-97.157,171.672,37.304,157.037
C06780=1048.646,216.929,-97.130,171.670,37.301,157.036
C06781=1048.639,216.680,-97.104,171.667,37.298,157.035
C06782=1048.633,216.432,-97.077,171.666,37.295,157.035
C06783=1048.626,216.183,-97.050,171.663,37.292,157.034
C06784=1048.620,215.935,-97.024,171.661,37.289,157.033
C06785=1048.613,215.686,-96.997,171.660,37.286,157.033
C06786=1048.607,215.438,-96.970,171.657,37.283,157.032
C06787=1048.601,215.189,-96.943,171.655,37.279,157.031
C06788=1048.594,214.941,-96.917,171.653,37.276,157.031
C06789=1048.588,214.692,-96.890,171.651,37.273,157.030
C06790=1048.582,214.444,-96.864,171.649,37.270,157.029
C06791=1048.575,214.195,-96.837,171.647,37.267,157.029
C06792=1048.569,213.947,-96.811,171.644,37.264,157.028
C06793=1048.562,213.698,-96.784,171.643,37.261,157.027
C06794=1048.556,213.450,-96.758,171.640,37.258,157.027
C06795=1048.549,213.201,-96.731,171.639,37.254,157.026
C06796=1048.544,212.953,-96.704,171.636,37.251,157.025
C06797=1048.536,212.704,-96.678,171.634,37.248,157.025
C06798=1048.531,212.455,-96.651,171.632,37.245,157.024
C06799=1048.524,212.207,-96.625,171.630,37.242,157.023
C06800=1048.518,211.958,-96.598,171.628,37.239,157.023
C06801=1048.511,211.710,-96.572,171.626,37.236,157.022
C06802=1048.504,211.462,-96.545,171.624,37.233,157.021
C06803=1048.498,211.213,-96.519,171.622,37.229,157.021
C06804=1048.491,210.964,-96.492,171.620,37.226,157.020
C06805=1048.486,210.716,-96.466,171.618,37.223,157.019
C06806=1048.478,210.467,-96.439,171.616,37.220,157.019
C06807=1048.472,210.219,-96.413,171.613,37.217,157.018
C06808=1048.466,209.971,-96.387,171.612,37.214,157.017
C06809=1048.459,209.722,-96.360,171.609,37.211,157.017
C06810=1048.453,209.474,-96.334,171.608,37.208,157.016
C06811=1048.446,209.224,-96.308,171.605,37.204,157.015
C06812=1048.440,208.976,-96.282,171.604,37.201,157.015
C06813=1048.433,208.728,-96.255,171.601,37.198,157.014
C06814=1048.427,208.479,-96.229,171.599,37.195,157.013
C06815=1048.421,208.231,-96.203,171.597,37.192,157.013
C06816=1048.413,207.983,-96.176,171.595,37.189,157.012
C06817=1048.408,207.734,-96.150,171.594,37.186,157.011
C06818=1048.401,207.485,-96.124,171.591,37.183,157.011
C06819=1048.394,207.222,-96.097,171.590,37.179,157.010
C06820=1048.387,206.960,-96.069,171.587,37.176,157.009
C06821=1048.381,206.697,-96.041,171.585,37.172,157.008
C06822=1048.373,206.434,-96.014,171.583,37.169,157.008
C06823=1048.347,205.382,-95.907,171.342,37.071,156.986
C06824=1048.341,205.134,-95.882,171.340,37.069,156.985
C06825=1048.336,204.885,-95.858,171.337,37.066,156.985
C06826=1048.330,204.636,-95.833,171.334,37.064,156.984
C06827=1048.323,204.388,-95.807,171.332,37.061,156.984
C06828=1048.317,204.139,-95.782,171.330,37.059,156.983
C06829=1048.311,203.890,-95.757,171.326,37.057,156.983
C06830=1048.306,203.642,-95.732,171.324,37.055,156.983
C06831=1048.299,203.393,-95.707,171.322,37.052,156.982
C06832=1048.294,203.144,-95.682,171.318,37.050,156.982
C06833=1048.287,202.895,-95.658,171.316,37.048,156.981
C06834=1048.280,202.647,-95.632,171.314,37.045,156.981
C06835=1048.275,202.398,-95.608,171.310,37.043,156.980
C06836=1048.269,202.149,-95.583,171.308,37.040,156.980
C06837=1048.263,201.901,-95.557,171.306,37.038,156.979
C06838=1048.257,201.651,-95.533,171.303,37.036,156.979
C06839=1048.251,201.404,-95.508,171.300,37.034,156.978
C06840=1048.245,201.154,-95.483,171.298,37.031,156.978
C06841=1048.238,200.906,-95.458,171.295,37.029,156.977
C06842=1048.232,200.657,-95.434,171.292,37.027,156.977
C06843=1048.225,200.408,-95.409,171.290,37.025,156.976
C06844=1048.220,200.160,-95.385,171.287,37.022,156.976
C06845=1048.214,199.911,-95.359,171.285,37.020,156.975
C06846=1048.207,199.662,-95.335,171.282,37.018,156.975
C06847=1048.201,199.413,-95.310,171.279,37.016,156.974
C06848=1048.195,199.165,-95.286,171.277,37.013,156.974
C06849=1048.189,198.916,-95.261,171.274,37.012,156.974
C06850=1048.182,198.667,-95.237,171.272,37.009,156.973
C06851=1048.176,198.419,-95.212,171.269,37.007,156.973
C06852=1048.171,198.170,-95.187,171.267,37.005,156.972
C06853=1048.164,197.921,-95.163,171.264,37.003,156.972
C06854=1048.158,197.672,-95.138,171.261,37.000,156.971
C06855=1048.152,197.424,-95.114,171.259,36.998,156.971
C06856=1048.146,197.176,-95.089,171.257,36.996,156.970
C06857=1048.140,196.926,-95.064,171.253,36.994,156.970
C06858=1048.133,196.677,-95.040,171.251,36.992,156.969
C06859=1048.127,196.429,-95.015,171.249,36.989,156.969
C06860=1048.121,196.180,-94.991,171.246,36.987,156.968
C06861=1048.115,195.931,-94.967,171.243,36.985,156.968
C06862=1048.109,195.683,-94.942,171.241,36.983,156.967
C06863=1048.103,195.434,-94.918,171.239,36.981,156.967
C06864=1048.097,195.186,-94.894,171.236,36.979,156.967
C06865=1048.091,194.937,-94.869,171.233,36.976,156.966
C06866=1048.085,194.688,-94.844,171.231,36.974,156.966
C06867=1048.079,194.440,-94.820,171.228,36.972,156.965
C06868=1048.073,194.190,-94.796,171.226,36.970,156.965
C06869=1048.066,193.941,-94.772,171.223,36.968,156.964
C06870=1048.060,193.693,-94.747,171.220,36.965,156.964
C06871=1048.054,193.444,-94.723,171.218,36.964,156.963
C06872=1048.048,193.196,-94.699,171.216,36.961,156.963
C06873=1048.042,192.947,-94.675,171.214,36.959,156.962
C06874=1048.036,192.698,-94.650,171.210,36.957,156.962
C06875=1048.030,192.449,-94.626,171.208,36.955,156.962
C06876=1048.024,192.201,-94.601,171.206,36.953,156.961
C06877=1048.018,191.952,-94.577,171.203,36.950,156.961
C06878=1048.012,191.703,-94.553,171.201,36.948,156.960
C06879=1048.006,191.454,-94.528,171.198,36.946,156.960
C06880=1048.000,191.205,-94.504,171.195,36.944,156.959
C06881=1047.994,190.957,-94.480,171.193,36.942,156.959
C06882=1047.988,190.708,-94.456,171.191,36.939,156.958
C06883=1047.983,190.459,-94.432,171.189,36.937,156.958
C06884=1047.975,190.175,-94.404,171.185,36.935,156.957
C06885=1047.968,189.890,-94.376,171.183,36.932,156.957
C06886=1047.961,189.607,-94.349,171.180,36.930,156.956
C06887=1047.954,189.322,-94.321,171.177,36.927,156.956
C06888=1047.948,189.073,-94.297,171.175,36.926,156.956
C06889=1047.942,188.824,-94.273,171.172,36.923,156.955
C06890=1047.936,188.575,-94.248,171.169,36.921,156.955
C06891=1047.930,188.327,-94.225,171.167,36.919,156.954
C06892=1047.925,188.078,-94.201,171.165,36.917,156.954
C06893=1047.919,187.829,-94.176,171.163,36.915,156.953
C06894=1047.913,187.581,-94.152,171.160,36.912,156.953
C06895=1047.907,187.332,-94.128,171.158,36.911,156.952
C06896=1047.901,187.083,-94.104,171.155,36.908,156.952
C06897=1047.895,186.834,-94.080,171.152,36.906,156.952
C06898=1047.889,186.585,-94.056,171.150,36.904,156.951
C06899=1047.883,186.337,-94.032,171.148,36.901,156.951
C06900=1047.878,186.087,-94.008,171.145,36.900,156.950
C06901=1047.872,185.839,-93.984,171.143,36.897,156.950
C06902=1047.866,185.590,-93.960,171.141,36.895,156.949
C06903=1047.860,185.341,-93.936,171.139,36.893,156.949
C06904=1047.854,185.093,-93.912,171.135,36.891,156.948
C06905=1047.848,184.844,-93.888,171.133,36.889,156.948
C06906=1047.842,184.596,-93.864,171.131,36.887,156.948
C06907=1047.836,184.346,-93.840,171.128,36.885,156.947
C06908=1047.830,184.097,-93.817,171.126,36.883,156.947
C06909=1047.825,183.849,-93.792,171.124,36.880,156.946
C06910=1047.818,183.600,-93.768,171.122,36.878,156.946
C06911=1047.812,183.351,-93.745,171.119,36.877,156.945
C06912=1047.806,183.102,-93.721,171.116,36.875,156.945
C06913=1047.800,182.854,-93.698,171.114,36.872,156.945
C06914=1047.793,182.604,-93.675,171.112,36.871,156.944
C06915=1047.787,182.356,-93.651,171.109,36.869,156.944
C06916=1047.780,182.107,-93.627,171.107,36.867,156.944
C06917=1047.774,181.858,-93.604,171.105,36.865,156.943
C06918=1047.768,181.609,-93.580,171.103,36.863,156.943
C06919=1047.762,181.360,-93.557,171.100,36.861,156.942
C06920=1047.756,181.112,-93.534,171.097,36.859,156.942
C06921=1047.749,180.863,-93.510,171.095,36.857,156.942
C06922=1047.744,180.614,-93.487,171.093,36.855,156.941
C06923=1047.737,180.365,-93.463,171.090,36.853,156.941
C06924=1047.731,180.116,-93.440,171.088,36.851,156.940
C06925=1047.725,179.867,-93.416,171.086,36.849,156.940
C06926=1047.719,179.618,-93.393,171.083,36.847,156.939
C06927=1047.713,179.370,-93.369,171.081,36.845,156.939
C06928=1047.706,179.121,-93.346,171.078,36.843,156.939
C06929=1047.700,178.873,-93.323,171.076,36.842,156.938
C06930=1047.694,178.624,-93.300,171.074,36.840,156.938
C06931=1047.687,178.375,-93.276,171.071,36.837,156.937
C06932=1047.682,178.126,-93.253,171.069,36.836,156.937
C06933=1047.675,177.877,-93.229,171.067,36.834,156.937
C06934=1047.669,177.628,-93.206,171.064,36.832,156.936
C06935=1047.663,177.380,-93.182,171.062,36.830,156.936
C06936=1047.657,177.130,-93.159,171.060,36.828,156.935
C06937=1047.651,176.881,-93.136,171.058,36.826,156.935
C06938=1047.645,176.633,-93.112,171.055,36.824,156.935
C06939=1047.639,176.384,-93.090,171.052,36.822,156.934
C06940=1047.632,176.135,-93.066,171.050,36.820,156.934
C06941=1047.626,175.886,-93.043,171.048,36.819,156.934
C06942=1047.620,175.638,-93.020,171.045,36.816,156.933
C06943=1047.614,175.389,-92.996,171.043,36.814,156.933
C06944=1047.608,175.140,-92.973,171.041,36.812,156.932
C06945=1047.602,174.891,-92.950,171.039,36.811,156.932
C06946=1047.596,174.642,-92.926,171.036,36.809,156.932
C06947=1047.589,174.393,-92.904,171.034,36.806,156.931
C06948=1047.583,174.108,-92.877,171.032,36.805,156.931
C06949=1047.576,173.824,-92.850,171.029,36.802,156.930
C06950=1047.569,173.538,-92.824,171.026,36.800,156.930
C06951=1047.562,173.254,-92.797,171.024,36.798,156.929
C06952=1047.556,173.005,-92.774,171.022,36.796,156.929
C06953=1047.549,172.756,-92.751,171.020,36.794,156.929
C06954=1047.544,172.507,-92.728,171.017,36.792,156.928
C06955=1047.538,172.259,-92.705,171.014,36.790,156.928
C06956=1047.532,172.010,-92.682,171.012,36.788,156.927
C06957=1047.526,171.761,-92.659,171.010,36.786,156.927
C06958=1047.520,171.512,-92.636,171.007,36.785,156.927
C06959=1047.514,171.263,-92.613,171.005,36.783,156.926
C06960=1047.507,171.015,-92.590,171.003,36.780,156.926
C06961=1047.502,170.766,-92.567,171.001,36.778,156.925
C06962=1047.496,170.517,-92.544,170.998,36.777,156.925
C06963=1047.489,170.267,-92.520,170.996,36.775,156.925
C06964=1047.484,170.018,-92.497,170.994,36.773,156.924
C06965=1047.478,169.769,-92.474,170.992,36.771,156.924
C06966=1047.471,169.522,-92.451,170.989,36.769,156.923
C06967=1047.466,169.273,-92.428,170.987,36.767,156.923
C06968=1047.460,169.024,-92.406,170.985,36.765,156.923
C06969=1047.454,168.775,-92.383,170.983,36.763,156.922
C06970=1047.448,168.525,-92.359,170.980,36.761,156.922
C06971=1047.442,168.276,-92.336,170.978,36.760,156.922
C06972=1047.436,168.028,-92.314,170.976,36.757,156.921
C06973=1047.430,167.779,-92.291,170.974,36.755,156.921
C06974=1047.424,167.530,-92.268,170.971,36.754,156.920
C06975=1047.418,167.281,-92.245,170.969,36.752,156.920
C06976=1047.413,167.032,-92.222,170.967,36.750,156.920
C06977=1047.407,166.783,-92.199,170.965,36.748,156.919
C06978=1047.400,166.535,-92.176,170.963,36.746,156.919
C06979=1047.394,166.286,-92.153,170.961,36.744,156.918
C06980=1047.388,166.037,-92.130,170.959,36.742,156.918
C06981=1047.382,165.788,-92.107,170.957,36.740,156.918
C06982=1047.377,165.539,-92.084,170.954,36.738,156.917
C06983=1047.370,165.290,-92.062,170.952,36.736,156.917
C06984=1047.365,165.041,-92.039,170.950,36.735,156.917
C06985=1047.359,164.792,-92.016,170.948,36.733,156.916
C06986=1047.353,164.543,-91.994,170.945,36.730,156.916
C06987=1047.347,164.294,-91.971,170.943,36.729,156.915
C06988=1047.341,164.046,-91.948,170.941,36.727,156.915
C06989=1047.335,163.797,-91.925,170.939,36.725,156.915
C06990=1047.330,163.548,-91.902,170.936,36.723,156.914
C06991=1047.324,163.299,-91.879,170.934,36.721,156.914
C06992=1047.317,163.050,-91.857,170.932,36.719,156.913
C06993=1047.312,162.801,-91.834,170.930,36.717,156.913
C06994=1047.306,162.553,-91.811,170.927,36.715,156.913
C06995=1047.300,162.303,-91.789,170.925,36.713,156.912
C06996=1047.295,162.054,-91.766,170.924,36.711,156.912
C06997=1047.288,161.806,-91.744,170.922,36.710,156.912
C06998=1047.283,161.557,-91.721,170.920,36.708,156.911
C06999=1047.277,161.308,-91.698,170.917,36.706,156.911
C07000=1047.271,161.059,-91.675,170.915,36.703,156.910
C07001=1047.265,160.810,-91.653,170.913,36.702,156.910
C07002=1047.259,160.561,-91.630,170.911,36.700,156.910
C07003=1047.253,160.312,-91.607,170.908,36.698,156.909
C07004=1047.247,160.063,-91.585,170.906,36.696,156.909
C07005=1047.241,159.814,-91.563,170.904,36.694,156.908
C07006=1047.235,159.565,-91.540,170.902,36.692,156.908
C07007=1047.229,159.317,-91.518,170.899,36.691,156.908
C07008=1047.223,159.067,-91.496,170.897,36.689,156.907
C07009=1047.217,158.819,-91.473,170.895,36.688,156.907
C07010=1047.210,158.570,-91.451,170.893,36.686,156.907
C07011=1047.205,158.320,-91.429,170.892,36.684,156.906
C07012=1047.198,158.036,-91.403,170.888,36.681,156.906
C07013=1047.191,157.750,-91.378,170.886,36.680,156.906
C07014=1047.183,157.465,-91.352,170.884,36.678,156.905
C07015=1047.177,157.180,-91.327,170.881,36.675,156.905
C07016=1047.171,156.931,-91.304,170.879,36.674,156.904
C07017=1047.165,156.682,-91.282,170.877,36.672,156.904
C07018=1047.158,156.433,-91.260,170.875,36.670,156.904
C07019=1047.153,156.184,-91.238,170.873,36.669,156.903
C07020=1047.146,155.935,-91.215,170.870,36.667,156.903
C07021=1047.141,155.686,-91.193,170.868,36.665,156.903
C07022=1047.135,155.437,-91.171,170.866,36.663,156.902
C07023=1047.128,155.188,-91.149,170.864,36.661,156.902
C07024=1047.123,154.939,-91.126,170.862,36.659,156.901
C07025=1047.117,154.690,-91.104,170.860,36.658,156.901
C07026=1047.111,154.442,-91.083,170.858,36.656,156.901
C07027=1047.104,154.193,-91.061,170.856,36.654,156.900
C07028=1047.099,153.944,-91.038,170.854,36.652,156.900
C07029=1047.093,153.695,-91.016,170.851,36.651,156.900
C07030=1047.086,153.446,-90.994,170.849,36.649,156.899
C07031=1047.080,153.197,-90.972,170.847,36.647,156.899
C07032=1047.074,152.948,-90.949,170.845,36.645,156.899
C07033=1047.068,152.699,-90.928,170.843,36.644,156.898
C07034=1047.062,152.449,-90.906,170.841,36.642,156.898
C07035=1047.055,152.201,-90.884,170.839,36.640,156.898
C07036=1047.049,151.952,-90.862,170.837,36.638,156.897
C07037=1047.044,151.703,-90.839,170.835,36.637,156.897
C07038=1047.038,151.454,-90.818,170.832,36.635,156.897
C07039=1047.032,151.205,-90.796,170.830,36.633,156.896
C07040=1047.025,150.956,-90.774,170.828,36.631,156.896
C07041=1047.020,150.707,-90.752,170.826,36.629,156.895
C07042=1047.014,150.458,-90.730,170.824,36.628,156.895
C07043=1047.007,150.209,-90.708,170.822,36.626,156.895
C07044=1047.001,149.960,-90.686,170.820,36.624,156.895
C07045=1046.996,149.711,-90.665,170.818,36.623,156.894
C07046=1046.989,149.463,-90.642,170.816,36.621,156.894
C07047=1046.984,149.213,-90.620,170.814,36.619,156.893
C07048=1046.977,148.964,-90.599,170.811,36.617,156.893
C07049=1046.971,148.715,-90.577,170.809,36.615,156.893
C07050=1046.965,148.466,-90.555,170.808,36.614,156.892
C07051=1046.959,148.218,-90.533,170.806,36.612,156.892
C07052=1046.953,147.969,-90.512,170.803,36.610,156.892
C07053=1046.947,147.719,-90.490,170.801,36.609,156.891
C07054=1046.941,147.471,-90.468,170.799,36.607,156.891
C07055=1046.935,147.221,-90.445,170.797,36.605,156.891
C07056=1046.929,146.972,-90.424,170.795,36.604,156.890
C07057=1046.923,146.724,-90.403,170.792,36.602,156.890
C07058=1046.917,146.474,-90.381,170.791,36.600,156.890
C07059=1046.910,146.225,-90.360,170.789,36.598,156.889
C07060=1046.904,145.976,-90.338,170.787,36.597,156.889
C07061=1046.898,145.728,-90.316,170.785,36.595,156.889
C07062=1046.891,145.478,-90.294,170.782,36.593,156.888
C07063=1046.886,145.230,-90.273,170.780,36.591,156.888
C07064=1046.880,144.981,-90.251,170.778,36.590,156.888
C07065=1046.874,144.732,-90.230,170.777,36.588,156.887
C07066=1046.867,144.482,-90.208,170.775,36.586,156.887
C07067=1046.861,144.233,-90.186,170.772,36.585,156.887
C07068=1046.856,143.985,-90.165,170.770,36.583,156.886
C07069=1046.850,143.735,-90.144,170.768,36.581,156.886
C07070=1046.843,143.486,-90.122,170.766,36.580,156.886
C07071=1046.837,143.237,-90.100,170.765,36.578,156.885
C07072=1046.832,142.989,-90.079,170.762,36.577,156.885
C07073=1046.826,142.739,-90.057,170.760,36.575,156.885
C07074=1046.819,142.490,-90.036,170.758,36.573,156.884
C07075=1046.813,142.241,-90.014,170.756,36.571,156.884
C07076=1046.806,141.956,-89.990,170.754,36.569,156.884
C07077=1046.799,141.670,-89.964,170.751,36.567,156.883
C07078=1046.792,141.385,-89.940,170.749,36.565,156.883
C07079=1046.785,141.100,-89.916,170.747,36.564,156.882
C07080=1046.779,140.851,-89.894,170.745,36.562,156.882
C07081=1046.773,140.601,-89.872,170.742,36.560,156.882
C07082=1046.767,140.353,-89.851,170.740,36.559,156.882
C07083=1046.761,140.104,-89.830,170.739,36.557,156.881
C07084=1046.755,139.854,-89.809,170.737,36.555,156.881
C07085=1046.749,139.605,-89.787,170.735,36.553,156.880
C07086=1046.743,139.356,-89.766,170.732,36.552,156.880
C07087=1046.737,139.107,-89.744,170.730,36.550,156.880
C07088=1046.730,138.858,-89.723,170.729,36.548,156.879
C07089=1046.725,138.610,-89.702,170.727,36.546,156.879
C07090=1046.719,138.360,-89.680,170.725,36.545,156.879
C07091=1046.713,138.111,-89.659,170.722,36.543,156.878
C07092=1046.706,137.862,-89.638,170.720,36.541,156.878
C07093=1046.700,137.613,-89.617,170.718,36.540,156.878
C07094=1046.694,137.364,-89.595,170.717,36.538,156.878
C07095=1046.688,137.115,-89.574,170.715,36.536,156.877
C07096=1046.682,136.867,-89.553,170.713,36.535,156.877
C07097=1046.676,136.617,-89.532,170.710,36.533,156.877
C07098=1046.670,136.368,-89.510,170.708,36.532,156.876
C07099=1046.663,136.119,-89.490,170.707,36.530,156.876
C07100=1046.657,135.870,-89.468,170.705,36.528,156.876
C07101=1046.651,135.620,-89.447,170.703,36.527,156.875
C07102=1046.646,135.372,-89.426,170.700,36.525,156.875
C07103=1046.639,135.123,-89.405,170.698,36.524,156.875
C07104=1046.633,134.874,-89.383,170.697,36.522,156.874
C07105=1046.628,134.625,-89.363,170.695,36.520,156.874
C07106=1046.621,134.376,-89.342,170.693,36.519,156.874
C07107=1046.615,134.127,-89.320,170.690,36.517,156.873
C07108=1046.609,133.877,-89.299,170.688,36.516,156.873
C07109=1046.602,133.628,-89.278,170.687,36.514,156.873
C07110=1046.597,133.380,-89.257,170.685,36.512,156.872
C07111=1046.591,133.130,-89.236,170.683,36.511,156.872
C07112=1046.585,132.882,-89.216,170.680,36.509,156.872
C07113=1046.578,132.633,-89.194,170.679,36.507,156.871
C07114=1046.573,132.383,-89.173,170.677,36.506,156.871
C07115=1046.566,132.135,-89.152,170.675,36.504,156.871
C07116=1046.560,131.885,-89.131,170.673,36.502,156.870
C07117=1046.555,131.636,-89.110,170.670,36.501,156.870
C07118=1046.548,131.388,-89.089,170.669,36.499,156.870
C07119=1046.542,131.138,-89.068,170.667,36.497,156.869
C07120=1046.536,130.889,-89.048,170.665,36.496,156.869
C07121=1046.530,130.640,-89.027,170.663,36.494,156.869
C07122=1046.523,130.391,-89.006,170.662,36.493,156.869
C07123=1046.517,130.142,-88.986,170.659,36.491,156.868
C07124=1046.511,129.893,-88.964,170.657,36.490,156.868
C07125=1046.505,129.644,-88.944,170.655,36.488,156.868
C07126=1046.498,129.395,-88.923,170.653,36.486,156.867
C07127=1046.492,129.145,-88.902,170.652,36.485,156.867
C07128=1046.486,128.897,-88.881,170.649,36.483,156.867
C07129=1046.480,128.647,-88.860,170.647,36.481,156.866
C07130=1046.474,128.399,-88.840,170.645,36.480,156.866
C07131=1046.467,128.149,-88.819,170.643,36.478,156.866
C07132=1046.461,127.900,-88.799,170.642,36.477,156.866
C07133=1046.455,127.651,-88.778,170.640,36.475,156.865
C07134=1046.448,127.402,-88.758,170.637,36.474,156.865
C07135=1046.443,127.153,-88.736,170.635,36.472,156.865
C07136=1046.436,126.904,-88.716,170.634,36.471,156.864
C07137=1046.430,126.655,-88.696,170.632,36.469,156.864
C07138=1046.424,126.406,-88.674,170.630,36.467,156.864
C07139=1046.418,126.157,-88.654,170.628,36.466,156.863
C07140=1046.410,125.871,-88.630,170.625,36.464,156.863
C07141=1046.403,125.586,-88.607,170.623,36.462,156.863
C07142=1046.397,125.300,-88.584,170.621,36.460,156.862
C07143=1046.389,125.013,-88.560,170.619,36.459,156.862
C07144=1046.384,124.765,-88.538,170.617,36.457,156.862
C07145=1046.377,124.515,-88.518,170.615,36.455,156.861
C07146=1046.371,124.267,-88.498,170.613,36.454,156.861
C07147=1046.365,124.017,-88.477,170.611,36.452,156.861
C07148=1046.359,123.769,-88.457,170.609,36.451,156.861
C07149=1046.352,123.519,-88.436,170.608,36.449,156.860
C07150=1046.347,123.270,-88.416,170.605,36.447,156.860
C07151=1046.340,123.021,-88.395,170.603,36.446,156.860
C07152=1046.334,122.772,-88.375,170.601,36.444,156.859
C07153=1046.328,122.522,-88.354,170.600,36.443,156.859
C07154=1046.322,122.274,-88.334,170.598,36.441,156.859
C07155=1046.315,122.025,-88.313,170.596,36.440,156.858
C07156=1046.310,121.776,-88.292,170.593,36.438,156.858
C07157=1046.304,121.527,-88.272,170.592,36.437,156.858
C07158=1046.297,121.277,-88.252,170.590,36.435,156.857
C07159=1046.292,121.029,-88.231,170.588,36.433,156.857
C07160=1046.285,120.779,-88.210,170.587,36.432,156.857
C07161=1046.279,120.530,-88.190,170.584,36.430,156.856
C07162=1046.273,120.281,-88.170,170.582,36.429,156.856
C07163=1046.267,120.032,-88.150,170.580,36.427,156.856
C07164=1046.261,119.783,-88.130,170.579,36.426,156.856
C07165=1046.255,119.534,-88.109,170.577,36.424,156.855
C07166=1046.249,119.285,-88.088,170.575,36.422,156.855
C07167=1046.243,119.035,-88.068,170.572,36.421,156.855
C07168=1046.237,118.787,-88.048,170.571,36.419,156.854
C07169=1046.231,118.538,-88.027,170.569,36.418,156.854
C07170=1046.225,118.288,-88.007,170.567,36.416,156.854
C07171=1046.219,118.039,-87.987,170.566,36.414,156.853
C07172=1046.213,117.790,-87.965,170.563,36.413,156.853
C07173=1046.207,117.541,-87.945,170.561,36.411,156.853
C07174=1046.201,117.292,-87.925,170.559,36.410,156.853
C07175=1046.194,117.043,-87.905,170.558,36.408,156.852
C07176=1046.189,116.794,-87.884,170.556,36.406,156.852
C07177=1046.183,116.545,-87.864,170.554,36.405,156.852
C07178=1046.176,116.295,-87.844,170.552,36.403,156.851
C07179=1046.170,116.047,-87.824,170.550,36.401,156.851
C07180=1046.165,115.798,-87.804,170.548,36.400,156.851
C07181=1046.158,115.548,-87.783,170.547,36.398,156.850
C07182=1046.152,115.299,-87.763,170.545,36.396,156.850
C07183=1046.147,115.050,-87.743,170.542,36.395,156.850
C07184=1046.141,114.801,-87.722,170.540,36.393,156.849
C07185=1046.135,114.552,-87.703,170.539,36.391,156.849
C07186=1046.129,114.303,-87.683,170.537,36.390,156.849
C07187=1046.123,114.053,-87.662,170.535,36.388,156.848
C07188=1046.117,113.804,-87.642,170.534,36.386,156.848
C07189=1046.111,113.555,-87.622,170.531,36.385,156.848
C07190=1046.104,113.306,-87.601,170.529,36.383,156.847
C07191=1046.098,113.057,-87.581,170.528,36.382,156.847
C07192=1046.092,112.808,-87.561,170.526,36.380,156.847
C07193=1046.086,112.559,-87.541,170.524,36.379,156.847
C07194=1046.080,112.310,-87.521,170.522,36.378,156.846
C07195=1046.074,112.061,-87.502,170.520,36.376,156.846
C07196=1046.067,111.811,-87.482,170.518,36.375,156.846
C07197=1046.061,111.562,-87.462,170.516,36.373,156.845
C07198=1046.055,111.313,-87.442,170.515,36.372,156.845
C07199=1046.049,111.065,-87.422,170.513,36.370,156.845
C07200=1046.043,110.815,-87.401,170.511,36.368,156.845
C07201=1046.037,110.566,-87.382,170.509,36.367,156.844
C07202=1046.031,110.317,-87.362,170.507,36.365,156.844
C07203=1046.024,110.067,-87.342,170.505,36.363,156.844
C07204=1046.017,109.782,-87.320,170.503,36.362,156.843
C07205=1046.010,109.496,-87.297,170.501,36.360,156.843
C07206=1046.003,109.210,-87.274,170.499,36.358,156.843
C07207=1045.996,108.924,-87.251,170.496,36.357,156.842
C07208=1045.990,108.675,-87.231,170.495,36.355,156.842
C07209=1045.984,108.426,-87.211,170.493,36.353,156.842
C07210=1045.978,108.176,-87.192,170.491,36.352,156.842
C07211=1045.971,107.928,-87.172,170.489,36.351,156.841
C07212=1045.965,107.678,-87.152,170.487,36.349,156.841
C07213=1045.959,107.429,-87.132,170.485,36.348,156.841
